	//
	Peeker		   : CollectionPeeker_Mock<5>;
	CollectionName : T_MaxString;
	i			   : UDINT;
END_VAR
IF TestSuite.Test(__POUNAME()).ExecuteTest() THEN
	Expected			  := TRUE;
	CollectionName		  := 'Test Collection';
	ExpectedNames[1]	  := ComponentArray[9].Name;
	ExpectedNames[2]	  := ComponentArray[0].Name;
	ExpectedNames[3]	  := ComponentArray[1].Name;
	ExpectedNames[4]	  := ComponentArray[2].Name;
	ExpectedNames[5]	  := ComponentArray[3].Name;
	Peeker.CollectionName := CollectionName;
	Peeker.PeekCollection(AllComponents);
	Peeker.MoveUpOne := TRUE;
	NamesEqual		 := TRUE;
	FOR i := 1 TO 5 DO
		__QUERYINTERFACE(Peeker.Items[i], CurrentComponent);
		ActualNames[i] := CurrentComponent.Name;
		NamesEqual	   := NamesEqual AND ActualNames[i] = ExpectedNames[i];
	END_FOR

	Actual := Peeker.FirstItem = 10 AND Peeker.LastItem = 4 AND NamesEqual;
	TestSuite.Test(__POUNAME()).AssertEqual(Expected, Actual);
END_IF
END_METHOD

METHOD NoCollection
VAR
	Expected : BOOL;
	Actual	 : BOOL;

	//
	Peeker		   : CollectionPeeker_Mock<5>;
	CollectionName : T_MaxString;
END_VAR
IF TestSuite.Test(__POUNAME()).ExecuteTest() THEN
	Expected		   := TRUE;
	CollectionName	   := '';
	Peeker.MoveDownOne := TRUE;
	Peeker.MoveUpOne   := TRUE;
	Peeker.PageDown	   := TRUE;
	Peeker.PageUp	   := TRUE;
	Actual			   := Peeker.CollectionName = CollectionName;
	TestSuite.Test(__POUNAME()).AssertEqual(Expected, Actual);
END_IF
END_METHOD

METHOD PageDownOne
VAR
	Expected		 : BOOL;
	Actual			 : BOOL;
	NamesEqual		 : BOOL;
	ExpectedNames	 : ARRAY[1..5] OF STRING[5];
	ActualNames		 : ARRAY[1..5] OF STRING[5];
	CurrentComponent : I_Component;

	//
	Peeker		   : CollectionPeeker_Mock<5>;
	CollectionName : T_MaxString;
	i			   : UDINT;
END_VAR
IF TestSuite.Test(__POUNAME()).ExecuteTest() THEN
	Expected			  := TRUE;
	CollectionName		  := 'Test Collection';
	ExpectedNames[1]	  := ComponentArray[5].Name;
	ExpectedNames[2]	  := ComponentArray[6].Name;
	ExpectedNames[3]	  := ComponentArray[7].Name;
	ExpectedNames[4]	  := ComponentArray[8].Name;
	ExpectedNames[5]	  := ComponentArray[9].Name;
	Peeker.CollectionName := CollectionName;
	Peeker.PeekCollection(AllComponents);
	Peeker.PageDown := TRUE;
	NamesEqual		:= TRUE;
	FOR i := 1 TO 5 DO
		__QUERYINTERFACE(Peeker.Items[i], CurrentComponent);
		ActualNames[i] := CurrentComponent.Name;
		NamesEqual	   := NamesEqual AND ActualNames[i] = ExpectedNames[i];
	END_FOR

	Actual := Peeker.FirstItem = 6 AND Peeker.LastItem = 10 AND NamesEqual;
	TestSuite.Test(__POUNAME()).AssertEqual(Expected, Actual);
END_IF
END_METHOD

METHOD PageDownRollover
VAR
	Expected		 : BOOL;
	Actual			 : BOOL;
	NamesEqual		 : BOOL;
	ExpectedNames	 : ARRAY[1..5] OF STRING[5];
	ActualNames		 : ARRAY[1..5] OF STRING[5];
	CurrentComponent : I_Component;

	//
	Peeker		   : CollectionPeeker_Mock<5>;
	CollectionName : T_MaxString;
	i			   : UDINT;
END_VAR
IF TestSuite.Test(__POUNAME()).ExecuteTest() THEN
	Expected			  := TRUE;
	CollectionName		  := 'Test Collection';
	ExpectedNames[1]	  := ComponentArray[8].Name;
	ExpectedNames[2]	  := ComponentArray[9].Name;
	ExpectedNames[3]	  := ComponentArray[0].Name;
	ExpectedNames[4]	  := ComponentArray[1].Name;
	ExpectedNames[5]	  := ComponentArray[2].Name;
	Peeker.CollectionName := CollectionName;
	Peeker.PeekCollection(AllComponents);
	Peeker.FirstItem := 4;
	Peeker.PageDown	 := TRUE;
	NamesEqual		 := TRUE;
	FOR i := 1 TO 5 DO
		__QUERYINTERFACE(Peeker.Items[i], CurrentComponent);
		ActualNames[i] := CurrentComponent.Name;
		NamesEqual	   := NamesEqual AND ActualNames[i] = ExpectedNames[i];
	END_FOR

	Actual := Peeker.FirstItem = 9 AND Peeker.LastItem = 3 AND NamesEqual;
	TestSuite.Test(__POUNAME()).AssertEqual(Expected, Actual);
END_IF
END_METHOD

METHOD PageUpOne
VAR
	Expected		 : BOOL;
	Actual			 : BOOL;
	NamesEqual		 : BOOL;
	ExpectedNames	 : ARRAY[1..5] OF STRING[5];
	ActualNames		 : ARRAY[1..5] OF STRING[5];
	CurrentComponent : I_Component;

	//
	Peeker		   : CollectionPeeker_Mock<5>;
	CollectionName : T_MaxString;
	i			   : UDINT;
END_VAR
IF TestSuite.Test(__POUNAME()).ExecuteTest() THEN
	Expected			  := TRUE;
	CollectionName		  := 'Test Collection';
	ExpectedNames[1]	  := ComponentArray[1].Name;
	ExpectedNames[2]	  := ComponentArray[2].Name;
	ExpectedNames[3]	  := ComponentArray[3].Name;
	ExpectedNames[4]	  := ComponentArray[4].Name;
	ExpectedNames[5]	  := ComponentArray[5].Name;
	Peeker.CollectionName := CollectionName;
	Peeker.PeekCollection(AllComponents);
	Peeker.FirstItem := 7;
	Peeker.PageUp	 := TRUE;
	NamesEqual		 := TRUE;
	FOR i := 1 TO 5 DO
		__QUERYINTERFACE(Peeker.Items[i], CurrentComponent);
		ActualNames[i] := CurrentComponent.Name;
		NamesEqual	   := NamesEqual AND ActualNames[i] = ExpectedNames[i];
	END_FOR

	Actual := Peeker.FirstItem = 2 AND Peeker.LastItem = 6 AND NamesEqual;
	TestSuite.Test(__POUNAME()).AssertEqual(Expected, Actual);
END_IF
END_METHOD

METHOD PageUpRollOver
VAR
	Expected		 : BOOL;
	Actual			 : BOOL;
	NamesEqual		 : BOOL;
	ExpectedNames	 : ARRAY[1..5] OF STRING[5];
	ActualNames		 : ARRAY[1..5] OF STRING[5];
	CurrentComponent : I_Component;

	//
	Peeker		   : CollectionPeeker_Mock<5>;
	CollectionName : T_MaxString;
	i			   : UDINT;
END_VAR
IF TestSuite.Test(__POUNAME()).ExecuteTest() THEN
	Expected			  := TRUE;
	CollectionName		  := 'Test Collection';
	ExpectedNames[1]	  := ComponentArray[6].Name;
	ExpectedNames[2]	  := ComponentArray[7].Name;
	ExpectedNames[3]	  := ComponentArray[8].Name;
	ExpectedNames[4]	  := ComponentArray[9].Name;
	ExpectedNames[5]	  := ComponentArray[0].Name;
	Peeker.CollectionName := CollectionName;
	Peeker.PeekCollection(AllComponents);
	Peeker.FirstItem := 2;
	Peeker.PageUp	 := TRUE;
	NamesEqual		 := TRUE;
	FOR i := 1 TO 5 DO
		__QUERYINTERFACE(Peeker.Items[i], CurrentComponent);
		ActualNames[i] := CurrentComponent.Name;
		NamesEqual	   := NamesEqual AND ActualNames[i] = ExpectedNames[i];
	END_FOR

	Actual := Peeker.FirstItem = 7 AND Peeker.LastItem = 1 AND NamesEqual;
	TestSuite.Test(__POUNAME()).AssertEqual(Expected, Actual);
END_IF
END_METHOD

METHOD SetCollectionCheck
VAR
	Expected		 : BOOL;
	Actual			 : BOOL;
	NamesEqual		 : BOOL;
	ExpectedNames	 : ARRAY[1..5] OF STRING[5];
	ActualNames		 : ARRAY[1..5] OF STRING[5];
	CurrentComponent : I_Component;

	//
	Peeker		   : CollectionPeeker_Mock<5>;
	CollectionName : T_MaxString;
	i			   : UDINT;
END_VAR
IF TestSuite.Test(__POUNAME()).ExecuteTest() THEN
	Expected			  := TRUE;
	CollectionName		  := 'Test Collection';
	ExpectedNames[1]	  := ComponentArray[0].Name;
	ExpectedNames[2]	  := ComponentArray[1].Name;
	ExpectedNames[3]	  := ComponentArray[2].Name;
	ExpectedNames[4]	  := ComponentArray[3].Name;
	ExpectedNames[5]	  := ComponentArray[4].Name;
	Peeker.CollectionName := CollectionName;
	Peeker.PeekCollection(AllComponents);
	NamesEqual := TRUE;
	FOR i := 1 TO 5 DO
		__QUERYINTERFACE(Peeker.Items[i], CurrentComponent);
		ActualNames[i] := CurrentComponent.Name;
		NamesEqual	   := NamesEqual AND ActualNames[i] = ExpectedNames[i];
	END_FOR

	Actual := Peeker.CollectionName = CollectionName AND Peeker.Collection.Count = AllComponents.Count AND Peeker.FirstItem = 1 AND Peeker.LastItem = 5 AND NamesEqual;
	TestSuite.Test(__POUNAME()).AssertEqual(Expected, Actual);
END_IF
END_METHOD

METHOD SetFirstItem
VAR
	Expected		 : BOOL;
	Actual			 : BOOL;
	NamesEqual		 : BOOL;
	ExpectedNames	 : ARRAY[1..5] OF STRING[5];
	ActualNames		 : ARRAY[1..5] OF STRING[5];
	CurrentComponent : I_Component;

	//
	Peeker		   : CollectionPeeker_Mock<5>;
	CollectionName : T_MaxString;
	i			   : UDINT;
END_VAR
IF TestSuite.Test(__POUNAME()).ExecuteTest() THEN
	Expected			  := TRUE;
	CollectionName		  := 'Test Collection';
	ExpectedNames[1]	  := ComponentArray[4].Name;
	ExpectedNames[2]	  := ComponentArray[5].Name;
	ExpectedNames[3]	  := ComponentArray[6].Name;
	ExpectedNames[4]	  := ComponentArray[7].Name;
	ExpectedNames[5]	  := ComponentArray[8].Name;
	Peeker.CollectionName := CollectionName;
	Peeker.PeekCollection(AllComponents);
	Peeker.FirstItem := 5;
	NamesEqual		 := TRUE;
	FOR i := 1 TO 5 DO
		__QUERYINTERFACE(Peeker.Items[i], CurrentComponent);
		ActualNames[i] := CurrentComponent.Name;
		NamesEqual	   := NamesEqual AND ActualNames[i] = ExpectedNames[i];
	END_FOR

	Actual := Peeker.FirstItem = 5 AND Peeker.LastItem = 9 AND NamesEqual;
	TestSuite.Test(__POUNAME()).AssertEqual(Expected, Actual);
END_IF
END_METHOD

END_FUNCTION_BLOCK

// ---- _Mockups/CollectionPeeker/CollectionPeeker_Mock.TcPOU
FUNCTION_BLOCK CollectionPeeker_Mock
VAR_GENERIC CONSTANT
	PeekSize2 : UDINT := 5;
END_VAR
EXTENDS CollectionPeeker<PeekSize2>
VAR
END_VAR

PROPERTY Collection : I_Collection
GET
Collection := _Collection;
END_GET
END_PROPERTY

END_FUNCTION_BLOCK

// ---- UnitTests/Force/ForcibleBool_TEST.TcPOU
FUNCTION_BLOCK ForcibleBool_TEST
VAR
END_VAR

ForceOff();
ForceOn();
UnforcedOff();
UnforcedOn();

METHOD ForceOff
VAR
	Expected	 : BOOL;
	Actual		 : BOOL;
	ForcibleBool : ForcibleBool('');
END_VAR
IF TestSuite.Test(__POUNAME()).ExecuteTest() THEN
	Expected := FALSE;
	ForcibleBool.SetForceState(E_ForceState.ForceOff);
	ForcibleBool.Input := TRUE;
	Actual			   := ForcibleBool.Output;
	TestSuite.Test(__POUNAME()).AssertEqual(Expected, Actual);
END_IF
END_METHOD

METHOD ForceOn
VAR
	Expected	 : BOOL;
	Actual		 : BOOL;
	ForcibleBool : ForcibleBool('');
END_VAR
IF TestSuite.Test(__POUNAME()).ExecuteTest() THEN
	Expected := TRUE;
	ForcibleBool.SetForceState(E_ForceState.ForceOn);
	ForcibleBool.Input := FALSE;
	Actual			   := ForcibleBool.Output;
	TestSuite.Test(__POUNAME()).AssertEqual(Expected, Actual);
END_IF
END_METHOD

METHOD UnforcedOff
VAR
	Expected	 : BOOL;
	Actual		 : BOOL;
	ForcibleBool : ForcibleBool('');
END_VAR
IF TestSuite.Test(__POUNAME()).ExecuteTest() THEN
	Expected := FALSE;
	ForcibleBool.SetForceState(E_ForceState.Unforced);
	ForcibleBool.Input := FALSE;
	Actual			   := ForcibleBool.Output;
	TestSuite.Test(__POUNAME()).AssertEqual(Expected, Actual);
END_IF
END_METHOD

METHOD UnforcedOn
VAR
	Expected	 : BOOL;
	Actual		 : BOOL;
	ForcibleBool : ForcibleBool('');
END_VAR
IF TestSuite.Test(__POUNAME()).ExecuteTest() THEN
	Expected := TRUE;
	ForcibleBool.SetForceState(E_ForceState.Unforced);
	ForcibleBool.Input := TRUE;
	Actual			   := ForcibleBool.Output;
	TestSuite.Test(__POUNAME()).AssertEqual(Expected, Actual);
END_IF
END_METHOD

END_FUNCTION_BLOCK

// ---- UnitTests/Force/ForcibleInt_Test.TcPOU
FUNCTION_BLOCK ForcibleInt_Test
VAR
END_VAR

ForceOff();
ForceOn();
ForcibleAcceptsValue();
ForciblePassesUnforcedValue();

METHOD ForceOff
VAR
	Expected	 : INT;
	Actual		 : INT;
	Forcible : ForcibleInt('');
END_VAR
IF TestSuite.Test(__POUNAME()).ExecuteTest() THEN
	Expected := 0;
	Forcible.SetForceState(E_ForceState.ForceOff);
	Forcible.Input := 12;
	Actual	:= Forcible.Output;
	TestSuite.Test(__POUNAME()).AssertEqual(Expected, Actual);
END_IF
END_METHOD

METHOD ForceOn
VAR
	Expected	 : INT;
	Actual		 : INT;
	Forcible : ForcibleInt('');
END_VAR
IF TestSuite.Test(__POUNAME()).ExecuteTest() THEN
	Expected := 16;
	Forcible.ForceValue := 16;
	Forcible.SetForceState(E_ForceState.ForceOn);
	Forcible.Input := 23;
	Actual			   := Forcible.Output;
	TestSuite.Test(__POUNAME()).AssertEqual(Expected, Actual);
END_IF
END_METHOD

METHOD ForcibleAcceptsValue
VAR
	Expected	 : INT;
	Actual		 : INT;
	Forcible : ForcibleInt('');
END_VAR
IF TestSuite.Test(__POUNAME()).ExecuteTest() THEN
	Expected := 17;
	Forcible.ForceValue := Expected;
	Actual			   := Forcible.ForceValue;
	TestSuite.Test(__POUNAME()).AssertEqual(Expected, Actual);
END_IF
END_METHOD

METHOD ForciblePassesUnforcedValue
VAR
	Expected	 : INT;
	Actual		 : INT;
	Forcible : ForcibleInt('');
END_VAR
IF TestSuite.Test(__POUNAME()).ExecuteTest() THEN
	Expected := 16;
	Forcible.SetForceState(E_ForceState.Unforced);
	Forcible.Input := 16;
	Actual			   := Forcible.Output;
	TestSuite.Test(__POUNAME()).AssertEqual(Expected, Actual);
END_IF
END_METHOD

END_FUNCTION_BLOCK

// ---- UnitTests/Utilities/Utilities_TEST.TcPOU
FUNCTION_BLOCK Utilities_TEST
VAR
END_VAR

CompareLREALFalse();
CompareLREALTrue();
CompareModuloFalse();
CompareModuloTrue();
PercentToAnalogConversion();
AnalogScaleReturns0IfInMinGTInMax();
AnalogScaleReturns0IfOutMinGTOutMax();
AnalogScaleReturnsOutMaxIFValueGTInMax();
AnalogScaleReturnsOutMinIFValueLTInMin();
AnalogueScaleConvertsCorrectly();
CalibrateAppliesGainCorrectly();
CalibrateAppliesOffsetCorrectly();

METHOD AnalogScaleReturns0IfInMinGTInMax
VAR
	InputGeneric : LREAL;
	TestScale : AnalogScale;

	Expected : LREAL := 0.0;
	Actual	 : LREAL;
END_VAR
IF TestSuite.Test(__POUNAME()).ExecuteTest() THEN
	InputGeneric							   := 750;
	TestScale.InputMaximum	   := 100;
	TestScale.InputMinimum	   := 200;
	TestScale.OutputMaximum	   := 10;
	TestScale.OutputMinimum	   := -10;
	Actual									   := TestScale.Transform(InputGeneric);
	TestSuite.Test(__POUNAME()).AssertEqual(Expected, Actual);
END_IF
END_METHOD

METHOD AnalogScaleReturns0IfOutMinGTOutMax
VAR
	InputGeneric : LREAL;
	TestScale : AnalogScale;

	Expected : LREAL := 0.0;
	Actual	 : LREAL;
END_VAR
IF TestSuite.Test(__POUNAME()).ExecuteTest() THEN
	InputGeneric							   := 750;
	TestScale.InputMaximum	   := 100;
	TestScale.InputMinimum	   := -200;
	TestScale.OutputMaximum	   := 10;
	TestScale.OutputMinimum	   := 20;
	Actual									   := TestScale.Transform(InputGeneric);
	TestSuite.Test(__POUNAME()).AssertEqual(Expected, Actual);
END_IF
END_METHOD

METHOD AnalogScaleReturnsOutMaxIFValueGTInMax
VAR
	InputGeneric : LREAL;
	TestScale : AnalogScale;

	Expected : LREAL := -10.0;
	Actual	 : LREAL;
END_VAR
IF TestSuite.Test(__POUNAME()).ExecuteTest() THEN
	InputGeneric			   := -110;
	TestScale.InputMaximum	   := 100;
	TestScale.InputMinimum	   := -100;
	TestScale.OutputMaximum	   := 10;
	TestScale.OutputMinimum	   := -10;
	Actual									   := TestScale.Transform(InputGeneric);
	TestSuite.Test(__POUNAME()).AssertEqual(Expected, Actual);
END_IF
END_METHOD

METHOD AnalogScaleReturnsOutMinIFValueLTInMin
VAR
	InputGeneric : LREAL;
	TestScale : AnalogScale;

	Expected : LREAL := 10.0;
	Actual	 : LREAL;
END_VAR
IF TestSuite.Test(__POUNAME()).ExecuteTest() THEN
	InputGeneric			   := 110;
	TestScale.InputMaximum	   := 100;
	TestScale.InputMinimum	   := -100;
	TestScale.OutputMaximum	   := 10;
	TestScale.OutputMinimum	   := -10;
	Actual									   := TestScale.Transform(InputGeneric);
	TestSuite.Test(__POUNAME()).AssertEqual(Expected, Actual);
END_IF
END_METHOD

METHOD AnalogueScaleConvertsCorrectly
VAR
	InputGeneric : LREAL;
	TestScale : AnalogScale;

	Expected : LREAL;
	Actual	 : LREAL;
END_VAR
IF TestSuite.Test(__POUNAME()).ExecuteTest() THEN
	InputGeneric							   := 500;
	Expected								   := 5;
	TestScale.InputMaximum	   := 1000;
	TestScale.InputMinimum	   := 0.0;
	TestScale.OutputMaximum	   := 10;
	TestScale.OutputMinimum	   := 0.0;
	Actual									   := TestScale.Transform(InputGeneric);
	TestSuite.Test(__POUNAME()).AssertEqual(Expected, Actual);
END_IF
END_METHOD

METHOD CalibrateAppliesGainCorrectly
VAR
	InputGeneric : LREAL;
	TestCalib : Calibrate;

	Expected : LREAL;
	Actual	 : LREAL;
END_VAR
IF TestSuite.Test(__POUNAME()).ExecuteTest() THEN
	InputGeneric							   := 500;
	Expected								   := 501;
	TestCalib.Gain	   := 1;
	TestCalib.Offset	   := 1.0;
	Actual									   := TestCalib.Transform(InputGeneric);
	TestSuite.Test(__POUNAME()).AssertEqual(Expected, Actual);
END_IF
END_METHOD

METHOD CalibrateAppliesOffsetCorrectly
VAR
	InputGeneric : LREAL;
	TestCalib : Calibrate;

	Expected : LREAL;
	Actual	 : LREAL;
END_VAR
IF TestSuite.Test(__POUNAME()).ExecuteTest() THEN
	InputGeneric							   := 500;
	Expected								   := 1000;
	TestCalib.Gain	   := 2;
	TestCalib.Offset	   := 0.0;
	Actual									   := TestCalib.Transform(InputGeneric);
	TestSuite.Test(__POUNAME()).AssertEqual(Expected, Actual);
END_IF
END_METHOD

METHOD CompareLREALFalse
VAR
	Expected : BOOL;
	Actual	 : BOOL;
END_VAR
IF TestSuite.Test(__POUNAME()).ExecuteTest() THEN
	Expected := FALSE;
	Actual	 := CompareLREAL(10.0, 11.8);
	TestSuite.Test(__POUNAME()).AssertEqual(Expected, Actual);
END_IF
END_METHOD

METHOD CompareLREALTrue
VAR
	Expected : BOOL;
	Actual	 : BOOL;
END_VAR
IF TestSuite.Test(__POUNAME()).ExecuteTest() THEN
	Expected := TRUE;
	Actual	 := CompareLREAL(10.5, 10.5);
	TestSuite.Test(__POUNAME()).AssertEqual(Expected, Actual);
END_IF
END_METHOD

METHOD CompareModuloFalse
VAR
	Expected : BOOL;
	Actual	 : BOOL;
END_VAR
IF TestSuite.Test(__POUNAME()).ExecuteTest() THEN
	Expected := FALSE;
	Actual	 := CompareModulo(360, 500);
	TestSuite.Test(__POUNAME()).AssertEqual(Expected, Actual);
END_IF
END_METHOD

METHOD CompareModuloTrue
VAR
	Expected : BOOL;
	Actual	 : BOOL;
END_VAR
IF TestSuite.Test(__POUNAME()).ExecuteTest() THEN
	Expected := TRUE;
	Actual	 := CompareModulo(0, 720);
	TestSuite.Test(__POUNAME()).AssertEqual(Expected, Actual);
END_IF
END_METHOD

METHOD PercentToAnalogConversion
VAR
	Expected : INT;
	Actual	 : INT;
END_VAR
IF TestSuite.Test(__POUNAME()).ExecuteTest() THEN
	Expected := 16383;
	Actual	 := PercentToAnalog(50);
	TestSuite.Test(__POUNAME()).AssertEqual(Expected, Actual);
END_IF
END_METHOD

END_FUNCTION_BLOCK

// ---- UnitTests/Digital/DigitalInput_NC_TEST.TcPOU
FUNCTION_BLOCK DigitalInput_NC_TEST
VAR
END_VAR

ForcedOn();
ForcedOff();
On();
Off();

METHOD ForcedOff : BOOL
VAR
	Expected		: BOOL;
	Actual			: BOOL;
	Input			: BOOL;
	DigitalInput_NC : DigitalInput_NC('DigitalInput', Input);
END_VAR
IF TestSuite.Test(__POUNAME()).ExecuteTest() THEN
	Expected			  := FALSE;
	DigitalInput_NC.Force := E_ForceState.ForceOff;
	Input				  := FALSE;
	Actual				  := DigitalInput_NC.IsActive;
	TestSuite.Test(__POUNAME()).AssertEqual(Expected, Actual);
END_IF
END_METHOD

METHOD ForcedOn : BOOL
VAR
	Expected		: BOOL;
	Actual			: BOOL;
	Input			: BOOL;
	DigitalInput_NC : DigitalInput_NC('DigitalInput', Input);
END_VAR
IF TestSuite.Test(__POUNAME()).ExecuteTest() THEN
	Expected			  := TRUE;
	DigitalInput_NC.Force := E_ForceState.ForceOn;
	Input				  := TRUE;
	Actual				  := DigitalInput_NC.IsActive;
	TestSuite.Test(__POUNAME()).AssertEqual(Expected, Actual);
END_IF
END_METHOD

METHOD Off : BOOL
VAR
	Expected		: BOOL;
	Actual			: BOOL;
	Input			: BOOL;
	DigitalInput_NC : DigitalInput_NC('DigitalInput', Input);
END_VAR
IF TestSuite.Test(__POUNAME()).ExecuteTest() THEN
	Expected			  := FALSE;
	DigitalInput_NC.Force := E_ForceState.Unforced;
	Input				  := TRUE;
	Actual				  := DigitalInput_NC.IsActive;
	TestSuite.Test(__POUNAME()).AssertEqual(Expected, Actual);
END_IF
END_METHOD

METHOD On
VAR
	Expected		: BOOL;
	Actual			: BOOL;
	Input			: BOOL;
	DigitalInput_NC : DigitalInput_NC('DigitalInput', Input);
END_VAR
IF TestSuite.Test(__POUNAME()).ExecuteTest() THEN
	Expected			  := TRUE;
	DigitalInput_NC.Force := E_ForceState.Unforced;
	Input				  := FALSE;
	Actual				  := DigitalInput_NC.IsActive;
	TestSuite.Test(__POUNAME()).AssertEqual(Expected, Actual);
END_IF
END_METHOD

END_FUNCTION_BLOCK

// ---- UnitTests/Digital/DigitalInput_NO_TEST.TcPOU
FUNCTION_BLOCK DigitalInput_NO_TEST
VAR
END_VAR

ForcedOn();
ForcedOff();
On();
Off();

METHOD ForcedOff : BOOL
VAR
	Expected		: BOOL;
	Actual			: BOOL;
	Input			: BOOL;
	DigitalInput_NO : DigitalInput_NO('DigitalInput', Input);
END_VAR
IF TestSuite.Test(__POUNAME()).ExecuteTest() THEN
	Expected			  := FALSE;
	DigitalInput_NO.Force := E_ForceState.ForceOff;
	Input				  := TRUE;
	Actual				  := DigitalInput_NO.IsActive;
	TestSuite.Test(__POUNAME()).AssertEqual(Expected, Actual);
END_IF
END_METHOD

METHOD ForcedOn : BOOL
VAR
	Expected		: BOOL;
	Actual			: BOOL;
	Input			: BOOL;
	DigitalInput_NO : DigitalInput_NO('DigitalInput', Input);
END_VAR
IF TestSuite.Test(__POUNAME()).ExecuteTest() THEN
	Expected			  := TRUE;
	DigitalInput_NO.Force := E_ForceState.ForceOn;
	Input				  := FALSE;
	Actual				  := DigitalInput_NO.IsActive;
	TestSuite.Test(__POUNAME()).AssertEqual(Expected, Actual);
END_IF
END_METHOD

METHOD Off : BOOL
VAR
	Expected		: BOOL;
	Actual			: BOOL;
	Input			: BOOL;
	DigitalInput_NO : DigitalInput_NO('DigitalInput', Input);
END_VAR
IF TestSuite.Test(__POUNAME()).ExecuteTest() THEN
	Expected			  := FALSE;
	DigitalInput_NO.Force := E_ForceState.Unforced;
	Input				  := FALSE;
	Actual				  := DigitalInput_NO.IsActive;
	TestSuite.Test(__POUNAME()).AssertEqual(Expected, Actual);
END_IF
END_METHOD

METHOD On
VAR
	Expected		: BOOL;
	Actual			: BOOL;
	Input			: BOOL;
	DigitalInput_NO : DigitalInput_NO('DigitalInput', Input);
END_VAR
IF TestSuite.Test(__POUNAME()).ExecuteTest() THEN
	Expected			  := TRUE;
	DigitalInput_NO.Force := E_ForceState.Unforced;
	Input				  := TRUE;
	Actual				  := DigitalInput_NO.IsActive;
	TestSuite.Test(__POUNAME()).AssertEqual(Expected, Actual);
END_IF
END_METHOD

END_FUNCTION_BLOCK

// ---- UnitTests/Digital/DigitalOutput_TEST.TcPOU
FUNCTION_BLOCK DigitalOutput_TEST
VAR
END_VAR

ForcedOn();
ForcedOff();
On();
Off();
ForceOffVisitor();
ForceOnVisitor();

METHOD ForcedOff
VAR
	Expected	  : BOOL;
	Actual		  : BOOL;
	Output		  : BOOL;
	DigitalOutput : DigitalOutput('Name', Output);
END_VAR
IF TestSuite.Test(__POUNAME()).ExecuteTest() THEN
	Expected			:= FALSE;
	DigitalOutput.Force := E_ForceState.ForceOff;
	DigitalOutput.On	:= TRUE;
	Actual				:= Output;
	TestSuite.Test(__POUNAME()).AssertEqual(Expected, Actual);
END_IF
END_METHOD

METHOD ForcedOn
VAR
	Expected	  : BOOL;
	Actual		  : BOOL;
	Output		  : BOOL;
	DigitalOutput : DigitalOutput('Name', Output);
END_VAR
IF TestSuite.Test(__POUNAME()).ExecuteTest() THEN
	Expected			:= TRUE;
	DigitalOutput.Force := E_ForceState.ForceOn;
	DigitalOutput.On	:= FALSE;
	Actual				:= Output;
	TestSuite.Test(__POUNAME()).AssertEqual(Expected, Actual);
END_IF
END_METHOD

METHOD ForceOffVisitor
VAR
	Expected	  : BOOL;
	Actual		  : BOOL;
	Output		  : BOOL;
	DigitalOutput : DigitalOutput('Name', Output);
	ForceVisitor  : ForceVisitor;
END_VAR
IF TestSuite.Test(__POUNAME()).ExecuteTest() THEN
	Expected			:= FALSE;
	DigitalOutput.Force := E_ForceState.ForceOn;
	ForceVisitor.Force	:= E_ForceState.ForceOff;
	DigitalOutput.Accept(ForceVisitor);
	DigitalOutput.On := TRUE;
	Actual			 := Output;
	TestSuite.Test(__POUNAME()).AssertEqual(Expected, Actual);
END_IF
END_METHOD

METHOD ForceOnVisitor
VAR
	Expected	  : BOOL;
	Actual		  : BOOL;
	Output		  : BOOL;
	DigitalOutput : DigitalOutput('Name', Output);
	ForceVisitor  : ForceVisitor;
END_VAR
IF TestSuite.Test(__POUNAME()).ExecuteTest() THEN
	Expected			:= TRUE;
	DigitalOutput.Force := E_ForceState.ForceOff;
	ForceVisitor.Force	:= E_ForceState.ForceOn;
	DigitalOutput.Accept(ForceVisitor);
	DigitalOutput.On := FALSE;
	Actual			 := Output;
	TestSuite.Test(__POUNAME()).AssertEqual(Expected, Actual);
END_IF
END_METHOD

METHOD Off : BOOL
VAR
	Expected	  : BOOL;
	Actual		  : BOOL;
	Output		  : BOOL;
	DigitalOutput : DigitalOutput('Name', Output);
END_VAR
IF TestSuite.Test(__POUNAME()).ExecuteTest() THEN
	Expected			:= FALSE;
	DigitalOutput.Force := E_ForceState.Unforced;
	DigitalOutput.On	:= FALSE;
	Actual				:= Output;
	TestSuite.Test(__POUNAME()).AssertEqual(Expected, Actual);
END_IF
END_METHOD

METHOD On
VAR
	Expected	  : BOOL;
	Actual		  : BOOL;
	Output		  : BOOL;
	DigitalOutput : DigitalOutput('Name', Output);
END_VAR
IF TestSuite.Test(__POUNAME()).ExecuteTest() THEN
	Expected			:= TRUE;
	DigitalOutput.Force := E_ForceState.Unforced;
	DigitalOutput.On	:= TRUE;
	Actual				:= Output;
	TestSuite.Test(__POUNAME()).AssertEqual(Expected, Actual);
END_IF
END_METHOD

END_FUNCTION_BLOCK

// ---- UnitTests/Digital/DigitalInput_Combiner_TEST.TcPOU
FUNCTION_BLOCK DigitalInput_Combiner_TEST
VAR
END_VAR

AddTwoInputsBothActiveCheckIsActive();
AddTwoInputsOneActiveCheckIsActiveFalse();
CheckIsActiveFalseWhenNoInputAdded();
TryAddDuplicateInput();

METHOD AddTwoInputsBothActiveCheckIsActive
VAR
	Expected			  : BOOL;
	Actual				  : BOOL;
	Input1				  : BOOL;
	Input2				  : BOOL;
	DigitalInput1		  : DigitalInput_NO('Input1', Input1);
	DigitalInput2		  : DigitalInput_NO('Input2', Input2);
	DigitalInput_Combiner : DigitalInput_Combiner<2>('Input1 & Input2');
END_VAR
IF TestSuite.Test(__POUNAME()).ExecuteTest() THEN
	Expected := TRUE;
	Input1	 := TRUE;
	Input2	 := TRUE;
	DigitalInput_Combiner.AddInput(DigitalInput1);
	DigitalInput_Combiner.AddInput(DigitalInput2);
	Actual := DigitalInput_Combiner.IsActive;
	TestSuite.Test(__POUNAME()).AssertEqual(Expected, Actual);
END_IF
END_METHOD

METHOD AddTwoInputsOneActiveCheckIsActiveFalse
VAR
	Expected			  : BOOL;
	Actual				  : BOOL;
	Input1				  : BOOL;
	Input2				  : BOOL;
	DigitalInput1		  : DigitalInput_NO('Input1', Input1);
	DigitalInput2		  : DigitalInput_NO('Input2', Input2);
	DigitalInput_Combiner : DigitalInput_Combiner<2>('Input1 & Input2');
END_VAR
IF TestSuite.Test(__POUNAME()).ExecuteTest() THEN
	Expected := FALSE;
	Input1	 := FALSE;
	Input2	 := TRUE;
	DigitalInput_Combiner.AddInput(DigitalInput1);
	DigitalInput_Combiner.AddInput(DigitalInput2);
	Actual := DigitalInput_Combiner.IsActive;
	TestSuite.Test(__POUNAME()).AssertEqual(Expected, Actual);
END_IF
END_METHOD

METHOD CheckIsActiveFalseWhenNoInputAdded
VAR
	Expected			  : BOOL;
	Actual				  : BOOL;
	DigitalInput_Combiner : DigitalInput_Combiner<2>('Input1 & Input2');
END_VAR
IF TestSuite.Test(__POUNAME()).ExecuteTest() THEN
	Expected := FALSE;
	Actual	 := DigitalInput_Combiner.IsActive;
	TestSuite.Test(__POUNAME()).AssertEqual(Expected, Actual);
END_IF
END_METHOD

METHOD TryAddDuplicateInput
VAR
	Expected			  : BOOL;
	Actual				  : BOOL;
	Input1				  : BOOL;
	Input2				  : BOOL;
	DigitalInput1		  : DigitalInput_NO('Input1', Input1);
	DigitalInput2		  : DigitalInput_NO('Input2', Input2);
	DigitalInput_Combiner : DigitalInput_Combiner<2>('Input1 & Input2');
END_VAR
IF TestSuite.Test(__POUNAME()).ExecuteTest() THEN
	Expected := FALSE;
	Input1	 := TRUE;
	Input2	 := FALSE;
	DigitalInput_Combiner.AddInput(DigitalInput1);
	DigitalInput_Combiner.AddInput(DigitalInput1);
	DigitalInput_Combiner.AddInput(DigitalInput2);
	Actual := DigitalInput_Combiner.IsActive;
	TestSuite.Test(__POUNAME()).AssertEqual(Expected, Actual);
END_IF
END_METHOD

END_FUNCTION_BLOCK

// ---- UnitTests/Digital/DigitalInput_Debounce_TEST.TcPOU
FUNCTION_BLOCK DigitalInput_Debounce_TEST
// DebounceRisingEdgeOn
VAR
	RisingEdgeOnExpected						: BOOL;
	RisingEdgeOnActual							: BOOL;
	RisingEdgeOnInput1							: BOOL;
	RisingEdgeOnDigitalInput1					: DigitalInput_NO('Input1', RisingEdgeOnInput1);
	RisingEdgeOnDigitalInput_DebounceRisingEdge : DigitalInput_DebounceRisingEdge('Input1', RisingEdgeOnDigitalInput1);
	RisingEdgeOnTestTimer						: TON;
END_VAR

// DebounceRisingEdgeStayOff
VAR
	RisingEdgeStayOffExpected						 : BOOL;
	RisingEdgeStayOffActual							 : BOOL;
	RisingEdgeStayOffInput1							 : BOOL;
	RisingEdgeStayOffDigitalInput1					 : DigitalInput_NO('Input1', RisingEdgeStayOffInput1);
	RisingEdgeStayOffDigitalInput_DebounceRisingEdge : DigitalInput_DebounceRisingEdge('Input1', RisingEdgeStayOffDigitalInput1);
	RisingEdgeStayOffTestTimer						 : TON;
END_VAR

// DebounceFallingEdgeOn
VAR
	FallingEdgeOnExpected						  : BOOL;
	FallingEdgeOnActual							  : BOOL;
	FallingEdgeOnInput1							  : BOOL := TRUE;
	FallingEdgeOnDigitalInput1					  : DigitalInput_NO('Input1', FallingEdgeOnInput1);
	FallingEdgeOnDigitalInput_DebounceFallingEdge : DigitalInput_DebounceFallingEdge('Input1', FallingEdgeOnDigitalInput1);
	FallingEdgeOnTestTimer						  : TON;
END_VAR

// DebounceFallingEdgeStayOff
VAR
	FallingEdgeStayOffExpected						   : BOOL;
	FallingEdgeStayOffActual						   : BOOL;
	FallingEdgeStayOffInput1						   : BOOL := TRUE;
	FallingEdgeStayOffDigitalInput1					   : DigitalInput_NO('Input1', FallingEdgeStayOffInput1);
	FallingEdgeStayOffDigitalInput_DebounceFallingEdge : DigitalInput_DebounceFallingEdge('Input1', FallingEdgeStayOffDigitalInput1);
	FallingEdgeStayOffTestTimer						   : TON;
END_VAR

DebounceRisingEdgeStayOff();
DebounceRisingEdgeOn();
DebounceFallingEdgeStayOff();
DebounceFallingEdgeOn();

METHOD DebounceFallingEdgeOn
VAR_INPUT
END_VAR
IF TestSuite.Test(__POUNAME()).ExecuteTest() THEN
	FallingEdgeOnExpected := TRUE;

	//
	FallingEdgeOnDigitalInput_DebounceFallingEdge.DebounceTime := T#250MS;
	FallingEdgeOnDigitalInput_DebounceFallingEdge.CyclicLogic();
	FallingEdgeOnInput1 := FALSE;

	//
	FallingEdgeOnTestTimer(IN := TRUE, PT := T#235MS);
	IF FallingEdgeOnTestTimer.Q THEN
		FallingEdgeOnActual := FallingEdgeOnDigitalInput_DebounceFallingEdge.IsActive;
		TestSuite.Test(__POUNAME()).AssertEqual(FallingEdgeOnExpected, FallingEdgeOnActual);
	END_IF
END_IF
END_METHOD

METHOD DebounceFallingEdgeStayOff
VAR_INPUT
END_VAR
IF TestSuite.Test(__POUNAME()).ExecuteTest() THEN
	FallingEdgeStayOffExpected := FALSE;

	//
	FallingEdgeStayOffDigitalInput_DebounceFallingEdge.DebounceTime := T#250MS;
	FallingEdgeStayOffDigitalInput_DebounceFallingEdge.CyclicLogic();
	FallingEdgeStayOffInput1 := FALSE;

	//
	FallingEdgeStayOffTestTimer(IN := TRUE, PT := T#265MS);
	IF FallingEdgeStayOffTestTimer.Q THEN
		FallingEdgeStayOffActual := FallingEdgeStayOffDigitalInput_DebounceFallingEdge.IsActive;
		TestSuite.Test(__POUNAME()).AssertEqual(FallingEdgeStayOffExpected, FallingEdgeStayOffActual);
	END_IF
END_IF
END_METHOD

METHOD DebounceRisingEdgeOn
IF TestSuite.Test(__POUNAME()).ExecuteTest() THEN
	RisingEdgeOnExpected := TRUE;
	RisingEdgeOnInput1	 := TRUE;

	//
	RisingEdgeOnDigitalInput_DebounceRisingEdge.DebounceTime := T#250MS;
	RisingEdgeOnDigitalInput_DebounceRisingEdge.CyclicLogic();

	//
	RisingEdgeOnTestTimer(IN := TRUE, PT := T#250MS);
	IF RisingEdgeOnTestTimer.Q THEN
		RisingEdgeOnActual := RisingEdgeOnDigitalInput_DebounceRisingEdge.IsActive;
		TestSuite.Test(__POUNAME()).AssertEqual(RisingEdgeOnExpected, RisingEdgeOnActual);
	END_IF
END_IF
END_METHOD

METHOD DebounceRisingEdgeStayOff
VAR_INPUT
END_VAR
IF TestSuite.Test(__POUNAME()).ExecuteTest() THEN
	RisingEdgeStayOffExpected := FALSE;
	RisingEdgeStayOffInput1	  := TRUE;

	//
	RisingEdgeStayOffDigitalInput_DebounceRisingEdge.DebounceTime := T#250MS;
	RisingEdgeStayOffDigitalInput_DebounceRisingEdge.CyclicLogic();

	//
	RisingEdgeStayOffTestTimer(IN := TRUE, PT := T#235MS);
	IF RisingEdgeStayOffTestTimer.Q THEN
		RisingEdgeStayOffActual := RisingEdgeStayOffDigitalInput_DebounceRisingEdge.IsActive;
		TestSuite.Test(__POUNAME()).AssertEqual(RisingEdgeStayOffExpected, RisingEdgeStayOffActual);
	END_IF
END_IF
END_METHOD

END_FUNCTION_BLOCK

// ---- UnitTests/Cylinder/Cylinder_TEST.TcPOU
FUNCTION_BLOCK Cylinder_TEST
VAR
	DiExtended		   : BOOL;
	DiRetracted		   : BOOL;
	DoExtend		   : BOOL;
	DoRetract		   : BOOL;
	Extend			   : DigitalOutput('Extend', DoExtend);
	Retract			   : DigitalOutput('Retract', DoRetract);
	Extended		   : DigitalInput_NO('Extended', DiExtended);
	Retracted		   : DigitalInput_NO('Retracted', DiRetracted);
	TestCylinder	   : Cylinder('Test Cylinder', Extend, Retract, Extended, Retracted) := (ExtendTimeout := T#250MS, RetractTimeout := T#250MS);
	TestCylinderEvents : Cylinder_TcEvents('Test Cylinder Events', TestCylinder);
	TonTimeout		   : TON;
END_VAR

RetractCheckRetracting();
RetractCheckRetracted();
ExtendCheckExtending();
ExtendCheckExtended();
ErrorBothSensorsOn();
ErrorRetracting();
ErrorExtending();

METHOD ErrorBothSensorsOn
VAR
	Expected : DINT;
	Actual	 : DINT;
END_VAR
IF TestSuite.Test(__POUNAME()).ExecuteTest() THEN
	Expected	:= 3;
	DiRetracted := TRUE;
	DiExtended	:= TRUE;
	TestCylinder.CyclicLogic();
	TestCylinderEvents.CyclicLogic();
	Actual := TestCylinderEvents.GetHighestActiveEventReaction();
	TestSuite.Test(__POUNAME()).AssertEqual(Expected, Actual);

	// Cleanup
	DiRetracted := FALSE;
	DiExtended	:= FALSE;
	TestCylinder.Reset();
	TestCylinderEvents.Reset();
	TestCylinder.CyclicLogic();
	TestCylinderEvents.CyclicLogic();
END_IF
END_METHOD

METHOD ErrorExtending
VAR
	Expected : DINT;
	Actual	 : DINT;
END_VAR
IF TestSuite.Test(__POUNAME()).ExecuteTest() THEN
	Expected	:= 3;
	DiRetracted := FALSE;
	DiExtended	:= FALSE;
	TestCylinder.Extend();
	TestCylinderEvents.CyclicLogic();
	TestCylinder.CyclicLogic();
	TonTimeout.IN := TRUE;
	IF TonTimeout.Q THEN
		Actual := TestCylinderEvents.GetHighestActiveEventReaction();
		TestSuite.Test(__POUNAME()).AssertEqual(Expected, Actual);

		// Cleanup
		TonTimeout.IN := FALSE;
		DiExtended	  := TRUE;
		TestCylinder.Reset();
		TestCylinderEvents.Reset();
		TestCylinderEvents.CyclicLogic();
		TestCylinder.CyclicLogic();
	END_IF
END_IF

TonTimeout(PT := T#300MS);
END_METHOD

METHOD ErrorRetracting
VAR
	Expected : DINT;
	Actual	 : DINT;
END_VAR
IF TestSuite.Test(__POUNAME()).ExecuteTest() THEN
	Expected	:= 3;
	DiRetracted := FALSE;
	DiExtended	:= FALSE;
	TestCylinder.Retract();
	TestCylinder.CyclicLogic();
	TestCylinderEvents.CyclicLogic();
	TonTimeout.IN := TRUE;
	IF TonTimeout.Q THEN
		Actual := TestCylinderEvents.GetHighestActiveEventReaction();
		TestSuite.Test(__POUNAME()).AssertEqual(Expected, Actual);

		// Cleanup
		TonTimeout.IN := FALSE;
		DiRetracted	  := TRUE;
		TestCylinder.Reset();
		TestCylinderEvents.Reset();
		TestCylinderEvents.CyclicLogic();
		TestCylinder.CyclicLogic();
	END_IF
END_IF

TonTimeout(PT := T#300MS);
END_METHOD

METHOD ExtendCheckExtended
VAR
	Expected : BOOL;
	Actual	 : BOOL;
END_VAR
IF TestSuite.Test(__POUNAME()).ExecuteTest() THEN
	Expected	:= TRUE;
	DiRetracted := FALSE;
	DiExtended	:= TRUE;
	TestCylinder.CyclicLogic();
	Actual := TestCylinder.Extended;
	TestSuite.Test(__POUNAME()).AssertEqual(Expected, Actual);
END_IF
END_METHOD

METHOD ExtendCheckExtending
VAR
	Expected : BOOL;
	Actual	 : BOOL;
END_VAR
IF TestSuite.Test(__POUNAME()).ExecuteTest() THEN
	Expected := TRUE;
	TestCylinder.Extend();
	TestCylinder.CyclicLogic();
	Actual := TestCylinder.Extending;
	TestSuite.Test(__POUNAME()).AssertEqual(Expected, Actual);
END_IF
END_METHOD

METHOD RetractCheckRetracted
VAR
	Expected : BOOL;
	Actual	 : BOOL;
END_VAR
IF TestSuite.Test(__POUNAME()).ExecuteTest() THEN
	Expected	:= TRUE;
	DiRetracted := TRUE;
	TestCylinder.CyclicLogic();
	Actual := TestCylinder.Retracted;
	TestSuite.Test(__POUNAME()).AssertEqual(Expected, Actual);
END_IF
END_METHOD

METHOD RetractCheckRetracting
VAR
	Expected : BOOL;
	Actual	 : BOOL;
END_VAR
IF TestSuite.Test(__POUNAME()).ExecuteTest() THEN
	Expected := TRUE;
	TestCylinder.Retract();
	TestCylinder.CyclicLogic();
	Actual := TestCylinder.Retracting;
	TestSuite.Test(__POUNAME()).AssertEqual(Expected, Actual);
END_IF
END_METHOD

END_FUNCTION_BLOCK

// ---- UnitTests/Safety/SafetyBase_TEST.TcPOU
FUNCTION_BLOCK SafetyBase_TEST
VAR
	ResetPulse : SafetyResetPulse('Reset');
	Group	   : SafetyGroup_TcEvents('Group');
	EStop_Sim  : SafetyEstopFB_TcEvents('E-Stop');
	EStop_OK   : SafetyEstopFB_TcEvents('E-Stop') := (ResetFunction := ResetPulse);
	EStop_NOK  : SafetyEstopFB_TcEvents('E-Stop') := (ResetFunction := ResetPulse);
END_VAR

VAR
	Init				  : BOOL := TRUE;
	InfoData_Group AT %Q* : ST_SafetyStateDiag;
	InfoData_OK	   AT %Q* : ST_SafetyStateDiag;
	InfoData_NOK   AT %Q* : ST_SafetyStateDiag;
	Run			   AT %I* : BOOL;
	Reset		   AT %I* : BOOL;
END_VAR

IF Init THEN
	InfoData_Group.State := E_SafetyGroup_State.Run;
	InfoData_OK.State	 := E_SafetyEStop_State.Run;
	InfoData_NOK.State	 := E_SafetyEStop_State.Error;
	Init				 := FALSE;
ELSE
	Group.CyclicLogic();
	EStop_OK.CyclicLogic();
	EStop_NOK.CyclicLogic();
	SimEstopOK();
	SimEstopOK();
	EstopOK();
	EstopNOK();
	GroupRun();
	EstopReset();
END_IF

METHOD EstopNOK
VAR_INST
	Expected : BOOL;
	Actual	 : BOOL;
END_VAR
IF TestSuite.Test(__POUNAME()).ExecuteTest() THEN
	Expected := FALSE;
	Actual	 := EStop_NOK.OK;
	TestSuite.Test(__POUNAME()).AssertEqual(Expected, Actual);
END_IF
END_METHOD

METHOD EstopOK
VAR_INST
	Expected : BOOL;
	Actual	 : BOOL;
END_VAR
IF TestSuite.Test(__POUNAME()).ExecuteTest() THEN
	Expected := TRUE;
	Actual	 := EStop_OK.OK;
	TestSuite.Test(__POUNAME()).AssertEqual(Expected, Actual);
END_IF
END_METHOD

METHOD EstopReset
VAR_INST
	Expected  : BOOL;
	Actual	  : BOOL;
	TestDelay : TON;
END_VAR
IF TestSuite.Test(__POUNAME()).ExecuteTest() THEN
	TestDelay(IN := TRUE, PT := T#50MS);
	Expected := TRUE;
	EStop_NOK.Reset();
	IF TestDelay.Q THEN
		Actual := Reset;
		TestSuite.Test(__POUNAME()).AssertEqual(Expected, Actual);
	END_IF
END_IF
END_METHOD

METHOD GroupRun
VAR_INST
	Expected : BOOL;
	Actual	 : BOOL;
END_VAR
IF TestSuite.Test(__POUNAME()).ExecuteTest() THEN
	Expected := TRUE;
	Actual	 := Run;
	TestSuite.Test(__POUNAME()).AssertEqual(Expected, Actual);
END_IF
END_METHOD

METHOD SimEstopNOK
VAR_INST
	Expected : BOOL;
	Actual	 : BOOL;
END_VAR
IF TestSuite.Test(__POUNAME()).ExecuteTest() THEN
	Expected := FALSE;
	EStop_Sim.SimulateSafetyState(E_SafetyEStop_State.Error);
	EStop_Sim.CyclicLogic();
	Actual := EStop_Sim.OK;
	TestSuite.Test(__POUNAME()).AssertEqual(Expected, Actual);
END_IF
END_METHOD

METHOD SimEstopOK
VAR_INST
	Expected : BOOL;
	Actual	 : BOOL;
END_VAR
IF TestSuite.Test(__POUNAME()).ExecuteTest() THEN
	Expected := TRUE;
	EStop_Sim.SimulateSafetyState(E_SafetyEStop_State.Run);
	EStop_Sim.CyclicLogic();
	Actual := EStop_Sim.OK;
	TestSuite.Test(__POUNAME()).AssertEqual(Expected, Actual);
END_IF
END_METHOD

END_FUNCTION_BLOCK

// ---- UnitTests/ADS/ADS_TEST.TcPOU
FUNCTION_BLOCK ADS_TEST
VAR
	AdsReadWrite		: AdsReadWrite('Ads Read/Write') := (AmsNetId := '', AmsPort := 851);
	AdsRwNumber AT %MD0 : UDINT							 := 50;
	AdsRwSymbol			: UDINT							 := 85;
	Value				: UDINT;
END_VAR

AdsRead();
AdsWrite();
AdsReadBySymbol();
AdsWriteBySymbol();
AdsReadWrite.CyclicLogic();

METHOD AdsRead
VAR_INST
	Expected : UDINT;
	Actual	 : UDINT;
	Seq		 : UDINT;
END_VAR
IF TestSuite.Test(__POUNAME()).ExecuteTest() THEN
	Expected := AdsRwNumber;
	CASE Seq OF
		0:
			AdsReadWrite.Read(IdxGrp	:= 16#4020,
							  IdxOffset := 16#0,
							  pDestAddr := ADR(Value),
							  Length	:= SIZEOF(Value));

			Seq := 10;

		10:
			IF NOT AdsReadWrite.Busy THEN
				Seq := 20;
			END_IF

		20:
			Actual := Value;
			TestSuite.Test(__POUNAME()).AssertEqual(Expected, Actual);
	END_CASE
END_IF
END_METHOD

METHOD AdsReadBySymbol
VAR_INST
	Expected : UDINT;
	Actual	 : UDINT;
	Seq		 : UDINT;
END_VAR
IF TestSuite.Test(__POUNAME()).ExecuteTest() THEN
	Expected := AdsRwSymbol;
	CASE Seq OF
		0:
			AdsReadWrite.ReadBySymbol(SymbolName := 'TestsBase.ADS_TEST.AdsRwSymbol', pDestAddr := ADR(Value), Length := SIZEOF(Value));
			Seq := 10;

		10:
			IF NOT AdsReadWrite.Busy THEN
				Seq := 20;
			END_IF

		20:
			Actual := Value;
			TestSuite.Test(__POUNAME()).AssertEqual(Expected, Actual);
	END_CASE
END_IF
END_METHOD

METHOD AdsWrite
VAR_INST
	Expected : UDINT;
	Actual	 : UDINT;
	Seq		 : UDINT;
END_VAR
IF TestSuite.Test(__POUNAME()).ExecuteTest() THEN
	Expected := 95;
	CASE Seq OF
		0:
			Value := 95;
			AdsReadWrite.Write(IdxGrp	   := 16#4020,
							   IdxOffset   := 16#0,
							   pSourceAddr := ADR(Value),
							   Length	   := SIZEOF(Value));

			Seq := 10;

		10:
			IF NOT AdsReadWrite.Busy THEN
				Seq := 20;
			END_IF

		20:
			Actual := AdsRwNumber;
			TestSuite.Test(__POUNAME()).AssertEqual(Expected, Actual);
	END_CASE
END_IF
END_METHOD

METHOD AdsWriteBySymbol
VAR_INST
	Expected : UDINT;
	Actual	 : UDINT;
	Seq		 : UDINT;
END_VAR
IF TestSuite.Test(__POUNAME()).ExecuteTest() THEN
	Expected := 79;
	CASE Seq OF
		0:
			Value := 79;
			AdsReadWrite.WriteBySymbol(SymbolName := 'TestsBase.ADS_TEST.AdsRwSymbol', pSourceAddr := ADR(Value), Length := SIZEOF(Value));
			Seq := 10;

		10:
			IF NOT AdsReadWrite.Busy THEN
				Seq := 20;
			END_IF

		20:
			Actual := AdsRwSymbol;
			TestSuite.Test(__POUNAME()).AssertEqual(Expected, Actual);
	END_CASE
END_IF
END_METHOD

END_FUNCTION_BLOCK

// ---- UnitTests/Digital/DigitalInput_ForceVisitor_TEST.TcPOU
FUNCTION_BLOCK DigitalInput_ForceVisitor_TEST
VAR
END_VAR

ForceOffVisitor_NO();
ForceOnVisitor_NO();
UnforcedVisitor_NO();
ForceOffVisitor_NC();
ForceOnVisitor_NC();
UnforcedVisitor_NC();

METHOD ForceOffVisitor_NC
VAR
	Expected	 : BOOL;
	Actual		 : BOOL;
	Input		 : BOOL;
	DigitalInput : DigitalInput_NC('DigitalInput', Input);
	ForceVisitor : ForceVisitor;
END_VAR
IF TestSuite.Test(__POUNAME()).ExecuteTest() THEN
	Expected		   := FALSE;
	DigitalInput.Force := E_ForceState.ForceOn;
	ForceVisitor.Force := E_ForceState.ForceOff;
	DigitalInput.Accept(ForceVisitor);
	Input  := FALSE;
	Actual := DigitalInput.IsActive;
	TestSuite.Test(__POUNAME()).AssertEqual(Expected, Actual);
END_IF
END_METHOD

METHOD ForceOffVisitor_NO
VAR
	Expected	 : BOOL;
	Actual		 : BOOL;
	Input		 : BOOL;
	DigitalInput : DigitalInput_NO('DigitalInput', Input);
	ForceVisitor : ForceVisitor;
END_VAR
IF TestSuite.Test(__POUNAME()).ExecuteTest() THEN
	Expected		   := FALSE;
	DigitalInput.Force := E_ForceState.ForceOn;
	ForceVisitor.Force := E_ForceState.ForceOff;
	DigitalInput.Accept(ForceVisitor);
	Input  := TRUE;
	Actual := DigitalInput.IsActive;
	TestSuite.Test(__POUNAME()).AssertEqual(Expected, Actual);
END_IF
END_METHOD

METHOD ForceOnVisitor_NC
VAR
	Expected	 : BOOL;
	Actual		 : BOOL;
	Input		 : BOOL;
	DigitalInput : DigitalInput_NC('DigitalInput', Input);
	ForceVisitor : ForceVisitor;
END_VAR
IF TestSuite.Test(__POUNAME()).ExecuteTest() THEN
	Expected		   := TRUE;
	DigitalInput.Force := E_ForceState.ForceOff;
	ForceVisitor.Force := E_ForceState.ForceOn;
	DigitalInput.Accept(ForceVisitor);
	Input  := FALSE;
	Actual := DigitalInput.IsActive;
	TestSuite.Test(__POUNAME()).AssertEqual(Expected, Actual);
END_IF
END_METHOD

METHOD ForceOnVisitor_NO
VAR
	Expected	 : BOOL;
	Actual		 : BOOL;
	Input		 : BOOL;
	DigitalInput : DigitalInput_NO('DigitalInput', Input);
	ForceVisitor : ForceVisitor;
END_VAR
IF TestSuite.Test(__POUNAME()).ExecuteTest() THEN
	Expected		   := TRUE;
	DigitalInput.Force := E_ForceState.ForceOff;
	ForceVisitor.Force := E_ForceState.ForceOn;
	DigitalInput.Accept(ForceVisitor);
	Input  := FALSE;
	Actual := DigitalInput.IsActive;
	TestSuite.Test(__POUNAME()).AssertEqual(Expected, Actual);
END_IF
END_METHOD

METHOD UnforcedVisitor_NC
VAR
	Expected	 : BOOL;
	Actual		 : BOOL;
	Input		 : BOOL;
	DigitalInput : DigitalInput_NC('DigitalInput', Input);
	ForceVisitor : ForceVisitor;
END_VAR
IF TestSuite.Test(__POUNAME()).ExecuteTest() THEN
	Expected		   := TRUE;
	DigitalInput.Force := E_ForceState.ForceOn;
	ForceVisitor.Force := E_ForceState.Unforced;
	DigitalInput.Accept(ForceVisitor);
	Input  := FALSE;
	Actual := DigitalInput.IsActive;
	TestSuite.Test(__POUNAME()).AssertEqual(Expected, Actual);
END_IF
END_METHOD

METHOD UnforcedVisitor_NO
VAR
	Expected	 : BOOL;
	Actual		 : BOOL;
	Input		 : BOOL;
	DigitalInput : DigitalInput_NO('DigitalInput', Input);
	ForceVisitor : ForceVisitor;
END_VAR
IF TestSuite.Test(__POUNAME()).ExecuteTest() THEN
	Expected		   := FALSE;
	DigitalInput.Force := E_ForceState.ForceOn;
	ForceVisitor.Force := E_ForceState.Unforced;
	DigitalInput.Accept(ForceVisitor);
	Input  := FALSE;
	Actual := DigitalInput.IsActive;
	TestSuite.Test(__POUNAME()).AssertEqual(Expected, Actual);
END_IF
END_METHOD

END_FUNCTION_BLOCK

// ---- UnitTests/Recipe/Recipe_TEST.TcPOU
FUNCTION_BLOCK Recipe_TEST
VAR
	ActiveRecipe	: ST_Recipe;
	UpdateRecipe	: ST_Recipe;
	RecipeManagment : RecipeManagment('Test Recipe Mgmt', nRecipe := SIZEOF(ST_Recipe), pActiveRecipeData := ADR(ActiveRecipe), pUpdateRecipeData := ADR(UpdateRecipe));
END_VAR

FirstCycleLoadNoChange();
DetectChangesLReal();
UpdateChangesLReal();
DetectChangesDint();
UpdateChangesDint();
DetectChangesBool();
UpdateChangesBool();
AutoLoad();

METHOD AutoLoad
VAR
	Expected : BOOL;
	Actual	 : BOOL;
END_VAR
IF TestSuite.Test(__POUNAME()).ExecuteTest() THEN
	Expected								:= TRUE;
	UpdateRecipe.ValueA						:= 0.756;
	RecipeManagment.AutoLoadChangesToActive := TRUE;
	RecipeManagment.CyclicLogic();
	Actual := NOT RecipeManagment.ChangesPending AND ActiveRecipe.ValueA = 0.756;
	TestSuite.Test(__POUNAME()).AssertEqual(Expected, Actual);
END_IF
END_METHOD

METHOD DetectChangesBool
VAR
	Expected : BOOL;
	Actual	 : BOOL;
END_VAR
IF TestSuite.Test(__POUNAME()).ExecuteTest() THEN
	Expected			:= TRUE;
	UpdateRecipe.ValueC := TRUE;
	RecipeManagment.CyclicLogic();
	Actual := RecipeManagment.ChangesPending;
	TestSuite.Test(__POUNAME()).AssertEqual(Expected, Actual);
END_IF
END_METHOD

METHOD DetectChangesDint
VAR
	Expected : BOOL;
	Actual	 : BOOL;
END_VAR
IF TestSuite.Test(__POUNAME()).ExecuteTest() THEN
	Expected			:= TRUE;
	UpdateRecipe.ValueB := 584;
	RecipeManagment.CyclicLogic();
	Actual := RecipeManagment.ChangesPending;
	TestSuite.Test(__POUNAME()).AssertEqual(Expected, Actual);
END_IF
END_METHOD

METHOD DetectChangesLReal
VAR
	Expected : BOOL;
	Actual	 : BOOL;
END_VAR
IF TestSuite.Test(__POUNAME()).ExecuteTest() THEN
	Expected			:= TRUE;
	UpdateRecipe.ValueA := 0.0584;
	RecipeManagment.CyclicLogic();
	Actual := RecipeManagment.ChangesPending;
	TestSuite.Test(__POUNAME()).AssertEqual(Expected, Actual);
END_IF
END_METHOD

METHOD FirstCycleLoadNoChange
VAR
	Expected : BOOL;
	Actual	 : BOOL;
END_VAR
IF TestSuite.Test(__POUNAME()).ExecuteTest() THEN
	Expected := FALSE;
	RecipeManagment.CyclicLogic();
	Actual := RecipeManagment.ChangesPending;
	TestSuite.Test(__POUNAME()).AssertEqual(Expected, Actual);
END_IF
END_METHOD

METHOD UpdateChangesBool
VAR
	Expected : BOOL;
	Actual	 : BOOL;
END_VAR
IF TestSuite.Test(__POUNAME()).ExecuteTest() THEN
	Expected := TRUE;
	RecipeManagment.LoadChangesToActive();
	RecipeManagment.CyclicLogic();
	Actual := NOT RecipeManagment.ChangesPending AND ActiveRecipe.ValueC;
	TestSuite.Test(__POUNAME()).AssertEqual(Expected, Actual);
END_IF
END_METHOD

METHOD UpdateChangesDint
VAR
	Expected : BOOL;
	Actual	 : BOOL;
END_VAR
IF TestSuite.Test(__POUNAME()).ExecuteTest() THEN
	Expected := TRUE;
	RecipeManagment.LoadChangesToActive();
	RecipeManagment.CyclicLogic();
	Actual := NOT RecipeManagment.ChangesPending AND ActiveRecipe.ValueB = 584;
	TestSuite.Test(__POUNAME()).AssertEqual(Expected, Actual);
END_IF
END_METHOD

METHOD UpdateChangesLReal
VAR
	Expected : BOOL;
	Actual	 : BOOL;
END_VAR
IF TestSuite.Test(__POUNAME()).ExecuteTest() THEN
	Expected := TRUE;
	RecipeManagment.LoadChangesToActive();
	RecipeManagment.CyclicLogic();
	Actual := NOT RecipeManagment.ChangesPending AND ActiveRecipe.ValueA = 0.0584;
	TestSuite.Test(__POUNAME()).AssertEqual(Expected, Actual);
END_IF
END_METHOD

END_FUNCTION_BLOCK

// ---- UnitTests/Analog/Analog_TEST.TcPOU
FUNCTION_BLOCK Analog_TEST
VAR
END_VAR

AnalogInputReturnsCorrectValue();
AnalogInputReturnsRawValueCorrectly();
AnalogOutputGenericCheckValue();
AnalogOutputGenericCheckRawValue();
AnalogAcceptsForceOff();
AnalogAcceptsForceOn();
AnalogAcceptsForceValue();
AnalogGenericPassesDataInValidCorrectly();
AnalogGenericPassesDataValidCorrectly();
AnalogGenericPassesErrorCorrectly();
AnalogGenericPassesOverrangeCorrectly();
AnalogGenericPassesUnderrangeCorrectly();

METHOD AnalogAcceptsForceOff
VAR
	InputGeneric		 : INT;
	AnalogInput_Generic	 : AnalogInput('Input Generic', InputGeneric);
	Expected : INT;
	Actual	 : INT;
END_VAR
IF TestSuite.Test(__POUNAME()).ExecuteTest() THEN
	Expected								   := 0;
	InputGeneric := 750;
	AnalogInput_Generic.ForceValue := 300;
	AnalogInput_Generic.Force := E_ForceState.ForceOff;
	Actual							:= AnalogInput_Generic.RawValue;
	TestSuite.Test(__POUNAME()).AssertEqual(Expected, Actual);
END_IF
END_METHOD

METHOD AnalogAcceptsForceOn
VAR
	InputGeneric		 : INT;
	AnalogInput_Generic	 : AnalogInput('Input Generic', InputGeneric);
	Expected : INT;
	Actual	 : INT;
END_VAR
IF TestSuite.Test(__POUNAME()).ExecuteTest() THEN
	Expected								   := 425;
	InputGeneric := 750;
	AnalogInput_Generic.ForceValue := Expected;
	AnalogInput_Generic.Force := E_ForceState.ForceOn;
	Actual							:= AnalogInput_Generic.RawValue;
	TestSuite.Test(__POUNAME()).AssertEqual(Expected, Actual);
END_IF
END_METHOD

METHOD AnalogAcceptsForceValue
VAR
	InputGeneric		 : INT;
	AnalogInput_Generic	 : AnalogInput('Input Generic', InputGeneric);
	Expected : INT;
	Actual	 : INT;
END_VAR
IF TestSuite.Test(__POUNAME()).ExecuteTest() THEN
	Expected								   := 750;
	AnalogInput_Generic.ForceValue := Expected;
	Actual							:= AnalogInput_Generic.ForceValue;
	TestSuite.Test(__POUNAME()).AssertEqual(Expected, Actual);
END_IF
END_METHOD

METHOD AnalogGenericPassesDataInValidCorrectly
VAR
	InputGeneric		 : INT;
	AnalogStatus : ST_AnalogInputStatus_Generic;
	AnalogInput_Generic	 : AnalogInput_Generic('Input Generic', InputGeneric, AnalogStatus );

	Expected : BOOL := TRUE;
	Actual	 : BOOL;
END_VAR
IF TestSuite.Test(__POUNAME()).ExecuteTest() THEN
	AnalogStatus.WcState := 0;
	Actual									   := AnalogInput_Generic.DataValid	;
	TestSuite.Test(__POUNAME()).AssertEqual(Expected, Actual);
END_IF
END_METHOD

METHOD AnalogGenericPassesDataValidCorrectly
VAR
	InputGeneric		 : INT;
	AnalogStatus : ST_AnalogInputStatus_Generic;
	AnalogInput_Generic	 : AnalogInput_Generic('Input Generic', InputGeneric, AnalogStatus );

	Expected : BOOL := FALSE;
	Actual	 : BOOL;
END_VAR
IF TestSuite.Test(__POUNAME()).ExecuteTest() THEN
	AnalogStatus.WcState := 1;
	Actual									   := AnalogInput_Generic.DataValid	;
	TestSuite.Test(__POUNAME()).AssertEqual(Expected, Actual);
END_IF
END_METHOD

METHOD AnalogGenericPassesErrorCorrectly
VAR
	InputGeneric		 : INT;
	AnalogStatus : ST_AnalogInputStatus_Generic;
	AnalogInput_Generic	 : AnalogInput_Generic('Input Generic', InputGeneric, AnalogStatus );

	Expected : BOOL := TRUE;
	Actual	 : BOOL;
END_VAR
IF TestSuite.Test(__POUNAME()).ExecuteTest() THEN
	AnalogStatus.Error := 1;
	Actual									   := AnalogInput_Generic.Error	;
	TestSuite.Test(__POUNAME()).AssertEqual(Expected, Actual);
END_IF
END_METHOD

METHOD AnalogGenericPassesOverrangeCorrectly
VAR
	InputGeneric		 : INT;
	AnalogStatus : ST_AnalogInputStatus_Generic;
	AnalogInput_Generic	 : AnalogInput_Generic('Input Generic', InputGeneric, AnalogStatus );

	Expected : BOOL := TRUE;
	Actual	 : BOOL;
END_VAR
IF TestSuite.Test(__POUNAME()).ExecuteTest() THEN
	AnalogStatus.Overrange := 1;
	Actual									   := AnalogInput_Generic.Overrange	;
	TestSuite.Test(__POUNAME()).AssertEqual(Expected, Actual);
END_IF
END_METHOD

METHOD AnalogGenericPassesUnderrangeCorrectly
VAR
	InputGeneric		 : INT;
	AnalogStatus : ST_AnalogInputStatus_Generic;
	AnalogInput_Generic	 : AnalogInput_Generic('Input Generic', InputGeneric, AnalogStatus );

	Expected : BOOL := TRUE;
	Actual	 : BOOL;
END_VAR
IF TestSuite.Test(__POUNAME()).ExecuteTest() THEN
	AnalogStatus.Underrrange := 1;
	Actual									   := AnalogInput_Generic.Underrange	;
	TestSuite.Test(__POUNAME()).AssertEqual(Expected, Actual);
END_IF
END_METHOD

METHOD AnalogInputReturnsCorrectValue
VAR
	InputGeneric		 : INT;
	AnalogInput_Generic	 : AnalogInput('Input Generic', InputGeneric);

	Expected : LREAL;
	Actual	 : LREAL;
END_VAR
IF TestSuite.Test(__POUNAME()).ExecuteTest() THEN
	InputGeneric							   := 8192;
	Expected								   := 6.00015;
	AnalogInput_Generic.Scale.InputMaximum	   := 32767;
	AnalogInput_Generic.Scale.InputMinimum	   := 0.0;
	AnalogInput_Generic.Scale.OutputMaximum	   := 10;
	AnalogInput_Generic.Scale.OutputMinimum	   := 0.0;
	AnalogInput_Generic.CalibrateLinear.Gain   := 2;
	AnalogInput_Generic.CalibrateLinear.Offset := 1;
	Actual									   := floor(AnalogInput_Generic.Value * 100000) / 100000;
	TestSuite.Test(__POUNAME()).AssertEqual(Expected, Actual);
END_IF
END_METHOD

METHOD AnalogInputReturnsRawValueCorrectly
VAR
	InputGeneric		 : INT;
	AnalogInput_Generic	 : AnalogInput('Input', InputGeneric);

	Expected : LREAL;
	Actual	 : LREAL;
END_VAR
IF TestSuite.Test(__POUNAME()).ExecuteTest() THEN
	InputGeneric							   := 750;
	Expected								   := 750;

	Actual									   := AnalogInput_Generic.RawValue;
	TestSuite.Test(__POUNAME()).AssertEqual(Expected, Actual);
END_IF
END_METHOD

METHOD AnalogOutputGenericCheckRawValue
VAR
	Expected : LREAL;
	Actual	 : LREAL;
	OutputGeneric		 : INT;
	AnalogOutput_Generic : AnalogOutput('Output Generic', OutputGeneric);
END_VAR
IF TestSuite.Test(__POUNAME()).ExecuteTest() THEN
	AnalogOutput_Generic.RawValue				:= 750;
	Expected									:= 750;
	AnalogOutput_Generic.Scale.InputMaximum		:= 10; // Process Value from plc e.g. liters
	AnalogOutput_Generic.Scale.InputMinimum		:= -10;
	AnalogOutput_Generic.Scale.OutputMaximum	:= 1000; // Output to terminal
	AnalogOutput_Generic.Scale.OutputMinimum	:= -1000;
	AnalogOutput_Generic.CalibrateLinear.Gain	:= 2;
	AnalogOutput_Generic.CalibrateLinear.Offset := 1;
	Actual										:= AnalogOutput_Generic.RawValue;
	TestSuite.Test(__POUNAME()).AssertEqual(Expected, Actual);
END_IF
END_METHOD

METHOD AnalogOutputGenericCheckValue
VAR
	Expected : LREAL;
	Actual	 : LREAL;
	OutputGeneric		 : INT;
	AnalogOutput_Generic : AnalogOutput('Output Generic', OutputGeneric);
END_VAR
IF TestSuite.Test(__POUNAME()).ExecuteTest() THEN
	Expected									:= 750;
	AnalogOutput_Generic.Scale.InputMaximum		:= 10; // Process Value from plc e.g. liters
	AnalogOutput_Generic.Scale.InputMinimum		:= -10;
	AnalogOutput_Generic.Scale.OutputMaximum	:= 1000; // Output to terminal
	AnalogOutput_Generic.Scale.OutputMinimum	:= -1000;
	AnalogOutput_Generic.CalibrateLinear.Gain	:= 1;
	AnalogOutput_Generic.CalibrateLinear.Offset := 0;
	AnalogOutput_Generic.Value					:= 7.5;
	Actual										:= AnalogOutput_Generic.RawValue;
	TestSuite.Test(__POUNAME()).AssertEqual(Expected, Actual);
END_IF
END_METHOD

END_FUNCTION_BLOCK

// ---- UnitTests/Serial/SerialConnection_Tests.TcPOU
FUNCTION_BLOCK SerialConnection_Tests
VAR
END_VAR

ByteConnectionAcceptsSendByte_Test();
StringConnectionAcceptsSendString_Test();
ByteConnectionRejectsSendByteWithNoLineCtrl_Test();
StringConnectionRejectsSendStringWithNoLineCtrl_Test();
ByteConnectionAcceptsSerialLineSet_Test();
ByteConnectionRejectsNulSerialLineSet_Test();
StringConnectionAcceptsSerialLineSet_Test();
StringConnectionRejectsNulSerialLineSet_Test();
ByteConnectionFlagsRecievedByte_Test();
ByteConnectionRecievesByteCorrectly_Test();
StringConnectionFlagsRecievedString_Test();
StringConnectionRecievesStringCorrectly_Test();
ByteConnectionRejectsResetWithNoLineCtrl_Test();
ByteConnectionResetsRxCommBuffer_Test();
StringConnectionRejectsResetWithNoLineCtrl_Test();
StringConnectionResetsRxCommBuffer_Test();

METHOD ByteConnectionAcceptsSendByte_Test : BOOL
VAR
	Expected : BOOL := TRUE;
	Actual	 : BOOL;
	seriallineCtrl : SerialLineControl_ADS;
	serialConnection : SerialByteConnection(Name := 'Channel 1',SerialLineController := seriallineCtrl);
END_VAR
IF TestSuite.Test(__POUNAME()).ExecuteTest() THEN
	Actual := SUCCEEDED(serialConnection.SendAByte(1));
	TestSuite.Test(__POUNAME()).AssertEqual(Expected, Actual);
END_IF
END_METHOD

METHOD ByteConnectionAcceptsSerialLineSet_Test : BOOL
VAR
	Expected : BOOL := TRUE;
	Actual	 : BOOL;
	seriallineCtrl : SerialLineControl_ADS;
	serialConnection : SerialByteConnection(Name := 'Channel 1',SerialLineController := 0);
END_VAR
IF TestSuite.Test(__POUNAME()).ExecuteTest() THEN
	Actual := serialConnection.SetDependencies(seriallineCtrl);
	TestSuite.Test(__POUNAME()).AssertEqual(Expected, Actual);
END_IF
END_METHOD

METHOD ByteConnectionFlagsRecievedByte_Test : BOOL
VAR
	Expected : BOOL := TRUE;
	Actual	 : BOOL;
	seriallineCtrl : MockSerialLineCtrl;
	serialConnection : SerialByteConnection(Name := 'Channel 1',SerialLineController := seriallineCtrl);
END_VAR
IF TestSuite.Test(__POUNAME()).ExecuteTest() THEN
	seriallineCtrl.SetComBufferByte(4);
	serialConnection.CyclicLogic();
	serialConnection.CyclicLogic();
	Actual := serialConnection.ByteDataRecieved;
	TestSuite.Test(__POUNAME()).AssertEqual(Expected, Actual);
END_IF
END_METHOD

METHOD ByteConnectionRecievesByteCorrectly_Test : BOOL
VAR
	Expected : BOOL := TRUE;
	Actual	 : BOOL;
	seriallineCtrl : MockSerialLineCtrl;
	serialConnection : SerialByteConnection(Name := 'Channel 1',SerialLineController := seriallineCtrl);
	TestByte : BYTE := 4;
END_VAR
IF TestSuite.Test(__POUNAME()).ExecuteTest() THEN
	seriallineCtrl.SetComBufferByte(TestByte);
	serialConnection.CyclicLogic();
	serialConnection.CyclicLogic();
	IF serialConnection.ByteDataRecieved THEN
		Actual := serialConnection.ByteData = TestByte;
	END_IF
	TestSuite.Test(__POUNAME()).AssertEqual(Expected, Actual);
END_IF
END_METHOD

METHOD ByteConnectionRejectsNulSerialLineSet_Test
VAR
	Expected : BOOL := FALSE;
	Actual	 : BOOL;
	serialConnection : SerialByteConnection(Name := 'Channel 1',SerialLineController := 0);
END_VAR
IF TestSuite.Test(__POUNAME()).ExecuteTest() THEN
	Actual := serialConnection.SetDependencies(0);
	TestSuite.Test(__POUNAME()).AssertEqual(Expected, Actual);
END_IF
END_METHOD

METHOD ByteConnectionRejectsResetWithNoLineCtrl_Test : BOOL
VAR
	Expected : BOOL := TRUE;
	Actual	 : BOOL;
	serialConnection : SerialByteConnection(Name := 'Channel 1',SerialLineController := 0);
END_VAR
IF TestSuite.Test(__POUNAME()).ExecuteTest() THEN
	Actual := FAILED(serialConnection.Reset());
	TestSuite.Test(__POUNAME()).AssertEqual(Expected, Actual);
END_IF
END_METHOD

METHOD ByteConnectionRejectsSendByteWithNoLineCtrl_Test : BOOL
VAR
	Expected : BOOL := TRUE;
	Actual	 : BOOL;
	serialConnection : SerialByteConnection(Name := 'Channel 1',SerialLineController := 0);
END_VAR
IF TestSuite.Test(__POUNAME()).ExecuteTest() THEN
	Actual := FAILED(serialConnection.SendAByte(1));
	TestSuite.Test(__POUNAME()).AssertEqual(Expected, Actual);
END_IF
END_METHOD

METHOD ByteConnectionResetsRxCommBuffer_Test : BOOL
VAR
	Expected : BOOL := TRUE;
	Actual	 : BOOL;
	seriallineCtrl : MockSerialLineCtrl;
	serialConnection : SerialByteConnection(Name := 'Channel 1',SerialLineController := seriallineCtrl);
END_VAR
IF TestSuite.Test(__POUNAME()).ExecuteTest() THEN
	seriallineCtrl.SetComBufferByte(4);
	serialConnection.CyclicLogic();
	serialConnection.CyclicLogic();
	serialConnection.Reset();
	Actual := seriallineCtrl.rxBuffer.RdIdx = 0;
	TestSuite.Test(__POUNAME()).AssertEqual(Expected, Actual);
END_IF
END_METHOD

METHOD StringConnectionAcceptsSendString_Test : BOOL
VAR
	Expected : BOOL := TRUE;
	Actual	 : BOOL;
	seriallineCtrl : SerialLineControl_ADS;
	serialConnection : SerialStringConnection(Name := 'Channel 1',SerialLineController := seriallineCtrl);
END_VAR
IF TestSuite.Test(__POUNAME()).ExecuteTest() THEN
	Actual := SUCCEEDED(serialConnection.SendAString('Bob'));
	TestSuite.Test(__POUNAME()).AssertEqual(Expected, Actual);
END_IF
END_METHOD

METHOD StringConnectionAcceptsSerialLineSet_Test : BOOL
VAR
	Expected : BOOL := TRUE;
	Actual	 : BOOL;
	seriallineCtrl : SerialLineControl_ADS;
	serialConnection : SerialStringConnection(Name := 'Channel 1',SerialLineController := 0);
END_VAR
IF TestSuite.Test(__POUNAME()).ExecuteTest() THEN
	Actual := serialConnection.SetDependencies(seriallineCtrl);
	TestSuite.Test(__POUNAME()).AssertEqual(Expected, Actual);
END_IF
END_METHOD

METHOD StringConnectionFlagsRecievedString_Test : BOOL
VAR
	Expected : BOOL := TRUE;
	Actual	 : BOOL;
	seriallineCtrl : MockSerialLineCtrl;
	serialConnection : SerialStringConnection(Name := 'Channel 1',SerialLineController := seriallineCtrl);
END_VAR
IF TestSuite.Test(__POUNAME()).ExecuteTest() THEN
	seriallineCtrl.SetComBufferString('$02 I Love Chips $03',20);
	serialConnection.SetSerialConfiguration('$02','$03');
	serialConnection.CyclicLogic();
	serialConnection.CyclicLogic();
	serialConnection.CyclicLogic();
	Actual := serialConnection.StringRecieved;
	TestSuite.Test(__POUNAME()).AssertEqual(Expected, Actual);
END_IF
END_METHOD

METHOD StringConnectionRecievesStringCorrectly_Test : BOOL
VAR
	Expected : BOOL := TRUE;
	Actual	 : BOOL;
	seriallineCtrl : MockSerialLineCtrl;
	serialConnection : SerialStringConnection(Name := 'Channel 1',SerialLineController := seriallineCtrl);
	testString : T_MaxString := '$02 I Love Chips $03';
END_VAR
IF TestSuite.Test(__POUNAME()).ExecuteTest() THEN
	seriallineCtrl.SetComBufferString('$02 I Love Chips $03',20);
	serialConnection.SetSerialConfiguration('$02','$03');
	serialConnection.CyclicLogic();
	serialConnection.CyclicLogic();
	serialConnection.CyclicLogic();
	IF serialConnection.StringRecieved THEN
		Actual := serialConnection.StringData = testString;
	END_IF
	TestSuite.Test(__POUNAME()).AssertEqual(Expected, Actual);
END_IF
END_METHOD

METHOD StringConnectionRejectsNulSerialLineSet_Test
VAR
	Expected : BOOL := FALSE;
	Actual	 : BOOL;
	serialConnection : SerialStringConnection(Name := 'Channel 1',SerialLineController := 0);
END_VAR
IF TestSuite.Test(__POUNAME()).ExecuteTest() THEN
	Actual := serialConnection.SetDependencies(0);
	TestSuite.Test(__POUNAME()).AssertEqual(Expected, Actual);
END_IF
END_METHOD

METHOD StringConnectionRejectsResetWithNoLineCtrl_Test : BOOL
VAR
	Expected : BOOL := TRUE;
	Actual	 : BOOL;
	serialConnection : SerialStringConnection(Name := 'Channel 1',SerialLineController := 0);
END_VAR
IF TestSuite.Test(__POUNAME()).ExecuteTest() THEN
	Actual := FAILED(serialConnection.Reset());
	TestSuite.Test(__POUNAME()).AssertEqual(Expected, Actual);
END_IF
END_METHOD

METHOD StringConnectionRejectsSendStringWithNoLineCtrl_Test : BOOL
VAR
	Expected : BOOL := TRUE;
	Actual	 : BOOL;
	serialConnection : SerialStringConnection(Name := 'Channel 1',SerialLineController := 0);
END_VAR
IF TestSuite.Test(__POUNAME()).ExecuteTest() THEN
	Actual := FAILED(serialConnection.SendAString('Bob'));
	TestSuite.Test(__POUNAME()).AssertEqual(Expected, Actual);
END_IF
END_METHOD

METHOD StringConnectionResetsRxCommBuffer_Test : BOOL
VAR
	Expected : BOOL := TRUE;
	Actual	 : BOOL;
	seriallineCtrl : MockSerialLineCtrl;
	serialConnection : SerialStringConnection(Name := 'Channel 1',SerialLineController := seriallineCtrl);
END_VAR
IF TestSuite.Test(__POUNAME()).ExecuteTest() THEN
	seriallineCtrl.SetComBufferByte(4);
	serialConnection.CyclicLogic();
	serialConnection.CyclicLogic();
	serialConnection.Reset();
	Actual := seriallineCtrl.rxBuffer.RdIdx = 0;
	TestSuite.Test(__POUNAME()).AssertEqual(Expected, Actual);
END_IF
END_METHOD

END_FUNCTION_BLOCK

// ---- _Mockups/SerialLineCtrl/MockSerialLineCtrl.TcPOU
FUNCTION_BLOCK MockSerialLineCtrl EXTENDS SerialLineControl_ADS
VAR
END_VAR

METHOD SetComBufferByte
VAR_INPUT
	ByteValue : BYTE;
END_VAR
rxComBuffer.Buffer[0] := ByteValue;
rxComBuffer.RdIdx := 0;
rxComBuffer.WrIdx := 0;
rxComBuffer.Count := 1;
rxComBuffer.FreeByte := 301;
END_METHOD

METHOD SetComBufferString
VAR_INPUT
	TestString : T_MaxString;
	StringSize : UINT;
END_VAR
VAR
	InterimString : T_MaxString;
	ByteOutput: ARRAY [0..Tc2_Utilities.MAX_STRING_LENGTH] OF BYTE;
	i : UDINT;
END_VAR
ByteOutput := MAXSTRING_TO_BYTEARR(TestString);
FOR i := StringSize - 1 TO MAX_STRING_LENGTH DO
	ByteOutput[i] := 0;
END_FOR
FOR i := 0 TO MAX_STRING_LENGTH DO
	rxComBuffer.Buffer[i] := ByteOutput[i];
END_FOR
rxComBuffer.RdIdx := 0;
rxComBuffer.WrIdx := 0;
rxComBuffer.Count := StringSize;
rxComBuffer.FreeByte := 301;
END_METHOD

END_FUNCTION_BLOCK

// ---- UnitTests/Axis/Axis_Test.TcPOU
FUNCTION_BLOCK Axis_Test
VAR
	AxisRef		: Tc2_MC2.AXIS_REF;
	Axis		: Mc2AxisPTP('Unit Test Axis', AxisRef) := (Override := 100.0);
	StartupTime : TON;
END_VAR

Axis.CyclicLogic();
StartupTime(IN := TRUE, PT := T#1S);
IF NOT StartupTime.Q THEN
	RETURN;
END_IF

Initialize();
Enable();
JogForward();
JogBackward();
MoveAbsoluteToStop();
Stop();
MoveAbsoluteToPoint();
Home();
Disable();
Error();
Reset();

METHOD Disable
VAR_INST
	Expected  : BOOL;
	Actual	  : BOOL;
	DoneTimer : TON;
END_VAR
IF TestSuite.Test(__POUNAME()).ExecuteTest() THEN
	Expected := TRUE;
	DoneTimer(IN := TRUE, PT := T#50MS);
	Axis.Disable();
	IF DoneTimer.Q THEN
		Actual := NOT Axis.Enabled AND NOT Axis.Busy AND NOT Axis.Error;
		TestSuite.Test(__POUNAME()).AssertEqual(Expected, Actual);
	END_IF
END_IF
END_METHOD

METHOD Enable
VAR_INST
	Expected  : BOOL;
	Actual	  : BOOL;
	DoneTimer : TON;
END_VAR
IF TestSuite.Test(__POUNAME()).ExecuteTest() THEN
	Expected := TRUE;
	DoneTimer(IN := TRUE, PT := T#50MS);
	Axis.Enable();
	IF DoneTimer.Q THEN
		Actual := Axis.Enabled AND NOT Axis.Busy AND NOT Axis.Error;
		TestSuite.Test(__POUNAME()).AssertEqual(Expected, Actual);
	END_IF
END_IF
END_METHOD

METHOD Error
VAR_INST
	Expected  : BOOL;
	Actual	  : BOOL;
	DoneTimer : TON;
END_VAR
IF TestSuite.Test(__POUNAME()).ExecuteTest() THEN
	Expected := TRUE;
	DoneTimer(IN := TRUE, PT := T#50MS);
	Axis.MoveAbsolute(20);
	IF DoneTimer.Q THEN
		Actual := (Axis.ErrorId <> 0) AND NOT Axis.Busy AND Axis.Error;
		TestSuite.Test(__POUNAME()).AssertEqual(Expected, Actual);
	END_IF
END_IF
END_METHOD

METHOD Home
VAR_INST
	Expected  : BOOL;
	Actual	  : BOOL;
	DoneTimer : TON;
	Command	  : BOOL := TRUE;
END_VAR
IF TestSuite.Test(__POUNAME()).ExecuteTest() THEN
	Expected := TRUE;
	DoneTimer(IN := TRUE, PT := T#100MS);
	IF Command AND NOT Axis.Busy THEN
		Command := FALSE;
		Axis.Home();
	END_IF

	IF DoneTimer.Q THEN
		Actual := CompareLREAL(Axis.ActualVelocity, 0, 0.1) AND CompareLREAL(Axis.ActualPosition, 0, 0.1) AND NOT Axis.Busy AND NOT Axis.Error;
		TestSuite.Test(__POUNAME()).AssertEqual(Expected, Actual);
	END_IF
END_IF
END_METHOD

METHOD Initialize
VAR_INST
	Expected  : BOOL;
	Actual	  : BOOL;
	DoneTimer : TON;
END_VAR
IF TestSuite.Test(__POUNAME()).ExecuteTest() THEN
	DoneTimer(IN := TRUE, PT := T#250MS);
	Expected := TRUE;
	IF DoneTimer.Q THEN
		Actual := Axis.Initialized AND NOT Axis.Error;
		TestSuite.Test(__POUNAME()).AssertEqual(Expected, Actual);
	END_IF
END_IF
END_METHOD

METHOD JogBackward
VAR_INST
	Expected  : BOOL;
	Actual	  : BOOL;
	DoneTimer : TON;
END_VAR
IF TestSuite.Test(__POUNAME()).ExecuteTest() THEN
	Expected := TRUE;
	DoneTimer(IN := TRUE, PT := T#1S);
	Axis.Jog(FALSE, TRUE);
	IF DoneTimer.Q THEN
		Actual := (Axis.ActualVelocity < 0) AND Axis.Busy AND NOT Axis.Error;
		TestSuite.Test(__POUNAME()).AssertEqual(Expected, Actual);
		Axis.Jog(FALSE, FALSE);
	END_IF
END_IF
END_METHOD

METHOD JogForward
VAR_INST
	Expected  : BOOL;
	Actual	  : BOOL;
	DoneTimer : TON;
END_VAR
IF TestSuite.Test(__POUNAME()).ExecuteTest() THEN
	Expected := TRUE;
	DoneTimer(IN := TRUE, PT := T#100MS);
	Axis.Jog(TRUE, FALSE);
	IF DoneTimer.Q THEN
		Actual := (Axis.ActualVelocity > 0) AND Axis.Busy AND NOT Axis.Error;
		TestSuite.Test(__POUNAME()).AssertEqual(Expected, Actual);
		Axis.Jog(FALSE, FALSE);
	END_IF
END_IF
END_METHOD

METHOD MoveAbsoluteToPoint
VAR_INST
	Expected  : BOOL;
	Actual	  : BOOL;
	DoneTimer : TON;
	Command	  : BOOL := TRUE;
END_VAR
IF TestSuite.Test(__POUNAME()).ExecuteTest() THEN
	Expected := TRUE;
	DoneTimer(IN := TRUE, PT := T#2S);
	IF Command AND NOT Axis.Busy THEN
		Command := FALSE;
		Axis.MoveAbsolute(100);
	END_IF

	IF DoneTimer.Q THEN
		Actual := CompareLREAL(Axis.ActualVelocity, 0, 0.1) AND CompareLREAL(Axis.ActualPosition, 100, 0.1) AND NOT Axis.Busy AND NOT Axis.Error;
		TestSuite.Test(__POUNAME()).AssertEqual(Expected, Actual);
	END_IF
END_IF
END_METHOD

METHOD MoveAbsoluteToStop
VAR_INST
	Expected  : BOOL;
	Actual	  : BOOL;
	DoneTimer : TON;
	Command	  : BOOL := TRUE;
END_VAR
IF TestSuite.Test(__POUNAME()).ExecuteTest() THEN
	Expected := TRUE;
	DoneTimer(IN := TRUE, PT := T#1S);
	IF Command AND NOT Axis.Busy THEN
		Command := FALSE;
		Axis.MoveAbsolute(1000);
	END_IF

	IF DoneTimer.Q THEN
		Actual := (Axis.ActualVelocity > 0) AND Axis.Busy AND NOT Axis.Error;
		TestSuite.Test(__POUNAME()).AssertEqual(Expected, Actual);
	END_IF
END_IF
END_METHOD

METHOD Reset
VAR_INST
	Expected  : BOOL;
	Actual	  : BOOL;
	DoneTimer : TON;
	Command	  : BOOL := TRUE;
END_VAR
IF TestSuite.Test(__POUNAME()).ExecuteTest() THEN
	Expected := TRUE;
	DoneTimer(IN := TRUE, PT := T#500MS);
	IF Command THEN
		Command := FALSE;
		Axis.Reset();
	END_IF

	IF DoneTimer.Q THEN
		Actual := (Axis.ErrorId = 0) AND NOT Axis.Busy AND NOT Axis.Error;
		TestSuite.Test(__POUNAME()).AssertEqual(Expected, Actual);
	END_IF
END_IF
END_METHOD

METHOD Stop
VAR_INST
	Expected  : BOOL;
	Actual	  : BOOL;
	DoneTimer : TON;
END_VAR
IF TestSuite.Test(__POUNAME()).ExecuteTest() THEN
	Expected := TRUE;
	DoneTimer(IN := TRUE, PT := T#500MS);
	Axis.Stop();
	IF DoneTimer.Q THEN
		Actual := CompareLREAL(Axis.ActualVelocity, 0, 0.1) AND NOT Axis.Busy AND NOT Axis.Error;
		TestSuite.Test(__POUNAME()).AssertEqual(Expected, Actual);
	END_IF
END_IF
END_METHOD

END_FUNCTION_BLOCK

// ---- UnitTests/EtherCat/EtherCatMaster_TEST.TcPOU
FUNCTION_BLOCK EtherCatMaster_TEST
VAR
	Provider : EtherCatEventProvider_Mockup('EtherCAT Event Provider');
	Master	 : EtherCatMaster_Mockup('EtherCAT Master Mock', EcStartupCycles := 1);
	Device	 : EtherCatIoDevice('Io Device');
	State	 : ST_EcExtendedSlaveState;
	Config	 : ST_EcSlaveConfigData;
END_VAR

IoDeviceStateFlags();
IoDeviceDiagnosticFlags();
IoDeviceCoeNullWithoutMailbox();
IoDeviceCoeWithMailbox();
MasterEventOncePerDevStateChange();
SlaveIndexByAddress();
SlaveIndexByAddressOutsideDenseRange();
SlaveRegistryNameAndHotConnect();
IoDeviceByAddrUsesMap();
AdsFailureKeepsErrorId();

// A failing slave state read aborts the sequence with ErrorSource Ads and the error id of the
// function block (or 16#745 on watchdog), never the former placeholder 999.
METHOD AdsFailureKeepsErrorId
VAR_INST
	Expected : BOOL;
	Actual	 : BOOL;
	Seq		 : UDINT;
	Cycles	 : UDINT;
END_VAR
IF TestSuite.Test(__POUNAME()).ExecuteTest() THEN
	Expected := TRUE;
	CASE Seq OF
		0:
			Master.LoadConfiguration(10);
			Master.SetMasterAmsNetId('1.2.3.4.5.6'); // no route: the read fails or times out
			Master.StartDiagnostic();
			Seq := 10;

		10:
			Master.RunSlaveState();
			Cycles := Cycles + 1;
			IF NOT Master.Busy OR Cycles > 2000 THEN
				Seq := 20;
			END_IF

		20:
			Actual := Master.Error AND (Master.ErrorSource = E_EcErrorSource.Ads) AND (Master.ErrorId <> 999) AND (Master.ErrorId <> 0);
			TestSuite.Test(__POUNAME()).AssertEqual(Expected, Actual);
	END_CASE
END_IF
END_METHOD

// The device returned for an address reflects the state of exactly that configured slave.
METHOD IoDeviceByAddrUsesMap
VAR_INST
	Expected : BOOL;
	Actual	 : BOOL;
END_VAR
IF TestSuite.Test(__POUNAME()).ExecuteTest() THEN
	Expected := TRUE;
	Master.LoadConfiguration(10);
	Master.SetSlaveState(Index := 2, DeviceState := 16#04, LinkState := 16#00); // slave at 1003 in SAFEOP
	Actual := Master.GetIoDeviceByAddr(1003).SafeOp AND Master.GetIoDeviceByAddr(1002).OP AND Master.GetIoDeviceByAddr(1004).OP AND NOT Master.GetIoDeviceByAddr(2000).OP;
	TestSuite.Test(__POUNAME()).AssertEqual(Expected, Actual);
END_IF
END_METHOD

METHOD IoDeviceCoeNullWithoutMailbox
VAR_INST
	Expected : STRING;
	Actual	 : STRING;
END_VAR
IF TestSuite.Test(__POUNAME()).ExecuteTest() THEN
	Expected			 := 'Null Terminal';
	Config.nMailboxInSize := 0;
	Device.Configuration REF= Config;
	Actual				 := Device.CoE.Name;
	TestSuite.Test(__POUNAME()).AssertEqual(Expected, Actual);
END_IF
END_METHOD

METHOD IoDeviceCoeWithMailbox
VAR_INST
	Expected : STRING;
	Actual	 : STRING;
END_VAR
IF TestSuite.Test(__POUNAME()).ExecuteTest() THEN
	Expected			 := 'CoE Terminal';
	Config.nMailboxInSize := 128;
	Config.nAddr		 := 1001;
	Device.Configuration REF= Config;
	Actual				 := Device.CoE.Name;
	TestSuite.Test(__POUNAME()).AssertEqual(Expected, Actual);
END_IF
END_METHOD

// deviceState bits 4..7 (error, invalid VPRS, init command error, disabled) are flags on top of the ESM state.
METHOD IoDeviceDiagnosticFlags
VAR_INST
	Expected : BOOL;
	Actual	 : BOOL;
END_VAR
IF TestSuite.Test(__POUNAME()).ExecuteTest() THEN
	Expected		  := TRUE;
	Device.State	 REF= State;
	State.deviceState := 16#F8; // OP with all four diagnostic bits set
	State.linkState	  := 16#00;
	Actual			  := Device.OP AND Device.DeviceError AND Device.InvalidVPRS AND Device.InitCmdError AND Device.Disabled;
	TestSuite.Test(__POUNAME()).AssertEqual(Expected, Actual);
END_IF
END_METHOD

METHOD IoDeviceStateFlags
VAR_INST
	Expected : BOOL;
	Actual	 : BOOL;
END_VAR
IF TestSuite.Test(__POUNAME()).ExecuteTest() THEN
	Expected		  := TRUE;
	Device.State	 REF= State;
	State.deviceState := 16#04; // SAFEOP, no diagnostic bits
	State.linkState	  := 16#00;
	Actual			  := Device.SafeOp AND NOT Device.OP AND NOT Device.PreOp AND NOT Device.Init AND NOT Device.Bootstrap
						 AND NOT Device.DeviceError AND NOT Device.InvalidVPRS AND NOT Device.InitCmdError AND NOT Device.Disabled;
	TestSuite.Test(__POUNAME()).AssertEqual(Expected, Actual);
END_IF
END_METHOD

// The MasterError event is raised once per DevState change, not every cycle the state persists.
METHOD MasterEventOncePerDevStateChange
VAR_INST
	Expected : UINT;
	Actual	 : UINT;
END_VAR
IF TestSuite.Test(__POUNAME()).ExecuteTest() THEN
	Expected := 1;
	Master.LoadConfiguration(10);
	Master.RegisterEventProvider(Provider);
	Master.SetMasterDevState(DevState := 16#0001, SlaveCount := 9); // link error, one slave missing
	Master.RunMasterState();
	Master.RunMasterState();
	Master.RunMasterState();
	Actual := Provider.MasterEventCount;
	TestSuite.Test(__POUNAME()).AssertEqual(Expected, Actual);
END_IF
END_METHOD

METHOD SlaveIndexByAddress
VAR_INST
	Expected : DINT;
	Actual	 : DINT;
END_VAR
IF TestSuite.Test(__POUNAME()).ExecuteTest() THEN
	Expected := 4;
	Master.LoadConfiguration(10);
	Actual := Master.GetSlaveIndexByAddr(1005);
	TestSuite.Test(__POUNAME()).AssertEqual(Expected, Actual);
END_IF
END_METHOD

// A user assigned address outside 1001.. is found by the linear fallback; unknown addresses give -1.
METHOD SlaveIndexByAddressOutsideDenseRange
VAR_INST
	Expected : BOOL;
	Actual	 : BOOL;
END_VAR
IF TestSuite.Test(__POUNAME()).ExecuteTest() THEN
	Expected := TRUE;
	Master.LoadConfiguration(10);
	Master.SetSlaveAddress(Index := 7, Addr := 60000);
	Actual := (Master.GetSlaveIndexByAddr(60000) = 7) AND (Master.GetSlaveIndexByAddr(1008) = -1) AND (Master.GetSlaveIndexByAddr(999) = -1);
	TestSuite.Test(__POUNAME()).AssertEqual(Expected, Actual);
END_IF
END_METHOD

// The master serves SyncUnitTask through I_EcSlaveRegistry: name and hot connect flag by index,
// safe defaults outside the configured range.
METHOD SlaveRegistryNameAndHotConnect
VAR_INST
	Expected : BOOL;
	Actual	 : BOOL;
	Registry : I_EcSlaveRegistry;
END_VAR
IF TestSuite.Test(__POUNAME()).ExecuteTest() THEN
	Expected := TRUE;
	Master.LoadConfiguration(10);
	Master.SetHotConnect(Index := 3);
	Registry := Master;
	Actual	 := (Registry.ConfiguredSlaveCount = 10)
				AND (Registry.GetSlaveName(4) = 'Slave5')
				AND Registry.IsHotConnectMember(3)
				AND NOT Registry.IsHotConnectMember(4)
				AND (Registry.GetSlaveName(10) = '')
				AND NOT Registry.IsHotConnectMember(10);
	TestSuite.Test(__POUNAME()).AssertEqual(Expected, Actual);
END_IF
END_METHOD

END_FUNCTION_BLOCK

// ---- _Mockups/EtherCat/EtherCatEventProvider_Mockup.TcPOU
// Counts the diagnostic events an EtherCatMaster raises instead of publishing TcEvents.
FUNCTION_BLOCK EtherCatEventProvider_Mockup EXTENDS Component IMPLEMENTS I_EtherCatDiagnosticEventProvider
VAR
	_MasterEventCount	: UINT;
	_SyncUnitEventCount : UINT;
	_ResetCount			: UINT;
	_LastEventId		: UDINT;
	_LastArgument1		: STRING;
	_LastArgument2		: STRING;
END_VAR

METHOD GetHighestActiveEventReaction : DINT
GetHighestActiveEventReaction := 0;
END_METHOD

METHOD GetHighestActiveEventSeverity : TcEventSeverity
GetHighestActiveEventSeverity := TcEventSeverity.Verbose;
END_METHOD

PROPERTY LastArgument1 : STRING
GET
LastArgument1 := _LastArgument1;
END_GET
END_PROPERTY

PROPERTY LastArgument2 : STRING
GET
LastArgument2 := _LastArgument2;
END_GET
END_PROPERTY

PROPERTY LastEventId : UDINT
GET
LastEventId := _LastEventId;
END_GET
END_PROPERTY

// Number of RaiseEtherCatDiagnosticEvent calls (master and slave events).
PROPERTY MasterEventCount : UINT
GET
MasterEventCount := _MasterEventCount;
END_GET
END_PROPERTY

METHOD RaiseEtherCatDiagnosticEvent
VAR_INPUT
	EventId	  : UDINT;
	Argument1 : STRING := '';
	Argument2 : STRING := '';
	Argument3 : STRING := '';
END_VAR
_MasterEventCount := _MasterEventCount + 1;
_LastEventId	  := EventId;
_LastArgument1	  := Argument1;
_LastArgument2	  := Argument2;
END_METHOD

METHOD RaiseSyncUnitEvent
VAR_INPUT
	EventId	  : UDINT;
	Argument1 : STRING := '';
	Argument2 : STRING := '';
	Argument3 : STRING := '';
END_VAR
_SyncUnitEventCount := _SyncUnitEventCount + 1;
_LastEventId		:= EventId;
_LastArgument1		:= Argument1;
_LastArgument2		:= Argument2;
END_METHOD

METHOD Reset
_ResetCount := _ResetCount + 1;
END_METHOD

PROPERTY ResetCount : UINT
GET
ResetCount := _ResetCount;
END_GET
END_PROPERTY

METHOD SetEventReactions
VAR_INPUT
	Verbose	 : DINT := 0;
	Info	 : DINT := 1;
	Warning	 : DINT := 2;
	Error	 : DINT := 3;
	Critical : DINT := 4;
END_VAR
END_METHOD

PROPERTY SyncUnitEventCount : UINT
GET
SyncUnitEventCount := _SyncUnitEventCount;
END_GET
END_PROPERTY

END_FUNCTION_BLOCK

// ---- _Mockups/EtherCat/EtherCatMaster_Mockup.TcPOU
// EtherCatMaster with its hardware inputs and slave arrays fed from the test instead of the master
// device. Exposes the protected evaluation steps so they can be driven without ADS or an EtherCAT master.
FUNCTION_BLOCK EtherCatMaster_Mockup EXTENDS EtherCatMaster<1, 1>
VAR
END_VAR

// Same inputs as EtherCatMaster.FB_Init; the base constructor receives them implicitly.
METHOD FB_Init : BOOL
VAR_INPUT
	bInitRetains	: BOOL; // TRUE: the retain variables are initialized (reset warm / reset cold)
	bInCopyCode		: BOOL; // TRUE: the instance will be copied to the copy code afterward (online change)
	Name			: T_MaxString;
	EcStartupCycles : UINT;
END_VAR
END_METHOD

// Current step of the slave diagnostic sequence (0 = idle).
PROPERTY DiagnosticStep : UDINT
GET
DiagnosticStep := SlaveSequence;
END_GET
END_PROPERTY

// Fakes a finished Initialize: Count slaves named Slave1..SlaveN at addresses 1001.., all OP, no mailbox.
METHOD LoadConfiguration
VAR_INPUT
	Count : UINT;
END_VAR

VAR
	i : UINT;
	n : UINT;
END_VAR
n := MIN(Count, MAX_EC_SLAVES + 1);

EcMaster.CfgSlaveCount := n;
EcMaster.SlaveCount	   := n;
SlaveCountUsed		   := n;

i := 0;
WHILE i < n DO
	ConfiguredSlaveInfo[i].nAddr		  := FIRST_SLAVE_ADDR + i;
	ConfiguredSlaveInfo[i].sName		  := CONCAT('Slave', TO_STRING(i + 1));
	ConfiguredSlaveInfo[i].nMailboxInSize := 0;
	SlavesState[i].deviceState			  := 16#08; // OP
	SlavesState[i].linkState			  := 16#00;
	SlaveTopologyInfo[i].nStatusBits	  := 0;	// no hot connect group (see SetHotConnect)
	IoDevice[i].Name					  := ConfiguredSlaveInfo[i].sName;
	IoDevice[i].State					  REF= SlavesState[i];
	IoDevice[i].Configuration			  REF= ConfiguredSlaveInfo[i];
	i									  := i + 1;
END_WHILE

BuildAddrToIndex();
Initialized := TRUE;
END_METHOD

// One evaluation of the master DevState (normally done by CyclicLogic).
METHOD RunMasterState : BOOL
RunMasterState := MasterState();
END_METHOD

// One cycle of the slave diagnostic sequence (normally done by CyclicLogic).
METHOD RunSlaveState
SlaveState();
_Busy := SlaveSequence <> 0;
END_METHOD

// Target of the diagnostic ADS reads (normally taken from EcMaster.AmsNetID in Initialize).
METHOD SetMasterAmsNetId
VAR_INPUT
	NetId : T_AmsNetId;
END_VAR
_MasterAmsNetId := NetId;
END_METHOD

// Fakes the master process image: DevState word and number of slaves currently on the bus.
METHOD SetMasterDevState
VAR_INPUT
	DevState   : UINT;
	SlaveCount : UINT;
END_VAR
EcMaster.DevState	:= DevState;
EcMaster.SlaveCount := SlaveCount;
END_METHOD

// Gives the configured slave Index another EtherCAT address and rebuilds the address map.
METHOD SetSlaveAddress
VAR_INPUT
	Index : UINT;
	Addr  : UINT;
END_VAR
ConfiguredSlaveInfo[Index].nAddr := Addr;
BuildAddrToIndex();
END_METHOD

// Fakes the topology read: marks one slave as member of a hot connect group.
METHOD SetHotConnect
VAR_INPUT
	Index : UINT;
END_VAR
SlaveTopologyInfo[Index].nStatusBits.4 := TRUE;
END_METHOD

// Fakes the state read of one slave.
METHOD SetSlaveState
VAR_INPUT
	Index		: UINT;
	DeviceState : BYTE;
	LinkState	: BYTE;
END_VAR
SlavesState[Index].deviceState := DeviceState;
SlavesState[Index].linkState   := LinkState;
END_METHOD

// Requests a slave diagnostic sequence (normally triggered by ChangeCount, slave count or frame WC state).
METHOD StartDiagnostic
RunSlaveDiag := TRUE;
END_METHOD

END_FUNCTION_BLOCK

// ---- UnitTests/AnyBuffer/AnyBuffer_TEST.TcPOU
PROGRAM AnyBuffer_TEST

// TEST_AnyBuffer_Clear();
// TEST_AnyBuffer_DeleteAtIndex();
// TEST_AnyBuffer_PeekAtIndex();
// TEST_AnyBuffer_ReplaceAtIndex();
// TEST_AnyBuffer_PushLeft();
// TEST_AnyBuffer_PushRight();
// TEST_AnyBuffer_PopLeft();
// TEST_AnyBuffer_PopRight();
// TEST_AnyBuffer_PopAtIndex();
// TEST_AnyBuffer_InsertAtIndex();

END_PROGRAM

// ---- _Mockups/AnyBuffer/Samples_AnyBuffer.TcPOU
PROGRAM Samples_AnyBuffer
(*
## Recent Performance Optimizations - Summary of Changes

### 1. FifoBuffer Optimization
**Changed from inefficient to efficient FIFO implementation:**
- **Before**: Used `AppendLeft` (O(n) - shifts all elements) for Push and `PopRight` (O(1)) for Pop
- **After**: Uses `AppendRight` (O(1) - no shifting) for Push and `PopLeft` (O(n)) for Pop
- **Benefit**: Push operations are now constant-time, which is much more common than Pop in FIFO queues
- **Performance**: Push now O(1) instead of O(n)
- **Documentation**: Updated all documentation to reflect the new behavior and performance characteristics

### 2. RingBuffer - Eliminated All Shifting Operations
**Implemented proper circular buffer with head/tail pointers:**
- **Added tracking variables**: `headIndex`, `tailIndex`, `elementCount`
- **Push**: Now uses circular indexing to overwrite oldest element **without any shifting** (true O(1))
- **Pop**: Uses `PeekAtIndex` with circular head pointer advancement **without shifting** (O(1))
- **Before**: Used `PopLeft()` which shifted all elements (O(n) operation)
- **After**: Direct circular buffer implementation with no shifting at all
- **Performance**: Both Push and Pop are now true O(1) constant-time operations

### 3. New WriteAtIndex Method in AnyBuffer
**Added low-level method for direct buffer access:**
- **Purpose**: Write to any physical index (0 to capacity-1) without changing buffer counters
- **Key difference from ReplaceAtIndex**:
  - `ReplaceAtIndex`: Only writes to logical indices (requires elements to exist)
  - `WriteAtIndex`: Writes to physical indices (works on empty buffer)
- **Use case**: Perfect for circular buffer implementations that manage their own counters
- **Documentation**: Comprehensive documentation with warnings about low-level nature

### 4. RingBuffer Updated to Use WriteAtIndex
- **Replaced** `ReplaceAtIndex` with `WriteAtIndex` for both initial fill and overwrite
- **Benefit**: No longer requires buffer to have elements, RingBuffer manages its own `elementCount`
- **Documentation**: Updated all RingBuffer documentation to reflect use of WriteAtIndex

### Performance Improvements Summary

| Operation | Before | After |
|-----------|--------|-------|
| **FifoBuffer.Push** | O(n) - shifts all | O(1) - append right |
| **FifoBuffer.Pop** | O(1) - no shift | O(n) - shift left |
| **RingBuffer.Push** | O(n) - PopLeft shifts | O(1) - direct write |
| **RingBuffer.Pop** | O(n) - PopLeft shifts | O(1) - PeekAtIndex |

**Result**: RingBuffer now implements a true circular buffer with optimal O(1) performance for all operations!

---

## Summary of Manual Test Programs

This project includes four manual test programs for interactively testing the AnyBuffer adapter
implementations. Each program provides control bits for manual testing and status monitoring.

### SampleFifo - Bounded Queue Testing
**File**: POUs/SampleFifo.TcPOU
**Adapter**: FifoBuffer (bounded FIFO queue without overwrite)
**Buffer Size**: 3 elements (indices 0..2)
**Performance**: Push O(1), Pop O(n)

**Configuration**:
```iecst
fifo : FifoBuffer(anyBuffer, overwrite := FALSE, reversed := FALSE);
```

**Features**:
- Tests bounded queue behavior (rejects push when full)
- Optimized for frequent Push operations (O(1) constant time)
- Status info: isEmpty, isFull, elementCount, capacity
- Operation counters: pushCount, popCount, pushFailCount, popFailCount
- Auto-incrementing element IDs for easy tracking

**Manual Controls**:
- `bPush` - Push new element (fails when buffer is full)
- `bPop` - Pop oldest element (FIFO order)
- `bClear` - Clear all elements

**Testing Scenario**:
1. Push 3 elements → buffer becomes full
2. Try pushing 4th element → fails (pushFailCount increments)
3. Pop 1 element → creates space
4. Push again → now succeeds

### SampleLifo - Bounded Stack Testing
**File**: POUs/SampleLifo.TcPOU
**Adapter**: LifoBuffer (bounded LIFO/stack without overwrite)
**Buffer Size**: 3 elements (indices 0..2)
**Performance**: Push O(1), Pop O(1)

**Configuration**:
```iecst
lifo : LifoBuffer(anyBuffer, overwrite := FALSE, reversed := FALSE);
```

**Features**:
- Tests bounded stack behavior (rejects push when full)
- LIFO semantics: Last-In, First-Out (stack operations)
- Both Push and Pop are O(1) constant time operations
- Status info: isEmpty, isFull, elementCount, capacity
- Operation counters: pushCount, popCount, pushFailCount, popFailCount
- Auto-incrementing element IDs for easy tracking

**Manual Controls**:
- `bPush` - Push new element to top of stack (fails when buffer is full)
- `bPop` - Pop most recent element (LIFO order)
- `bClear` - Clear all elements

**Testing Scenario**:
1. Push elements with IDs 1, 2, 3 → buffer becomes full
2. Try pushing 4th element → fails (pushFailCount increments)
3. Pop element → returns ID 3 (last pushed, LIFO)
4. Pop again → returns ID 2 (second-to-last pushed)
5. Pop again → returns ID 1 (first pushed)
6. Observe: LIFO behavior - reverse order from FIFO

### SampleRing - Circular Buffer Testing
**File**: POUs/SampleRing.TcPOU
**Adapter**: RingBuffer (circular buffer with automatic overwrite)
**Buffer Size**: 5 elements (indices 0..4)
**Performance**: Push O(1), Pop O(1) - **No shifting operations!**

**Configuration**:
```iecst
ring : RingBuffer(anyBuffer, overwriteEnabled := TRUE);
```

**Features**:
- Tests circular buffer behavior (automatic overwrite of oldest)
- True O(1) performance using head/tail circular indexing
- No element shifting - direct memory access with WriteAtIndex
- Status info: isEmpty, isFull, elementCount, capacity, overwriteEnabled
- Operation counters: pushCount, popCount, pushFailCount, popFailCount, **overwriteCount**
- Buffer snapshot array for visualizing circular behavior
- Tracks how many times push triggered an overwrite

**Manual Controls**:
- `bPush` - Push new element (overwrites oldest when full)
- `bPop` - Pop oldest element
- `bClear` - Clear all elements
- `bToggleOverwrite` - Display toggle (informational only)

**Testing Scenario**:
1. Push 5 elements → buffer becomes full: [0, 1, 2, 3, 4]
2. Push 6th element (ID=5) → succeeds, removes 0: [1, 2, 3, 4, 5]
3. Push 7th element (ID=6) → succeeds, removes 1: [2, 3, 4, 5, 6]
4. Watch bufferSnapshot to observe elements cycling through
5. Pop retrieves current oldest (not original first element)

### SampleList - Directional Fill with Shift-Overwrite
**File**: POUs/SampleList.TcPOU
**Adapter**: List (configurable-direction FIFO with shift-overwrite)
**Buffer Size**: 5 elements (indices 0..4)

**Configuration**:
```iecst
list : List(anyBuffer, fillFromLeft := FALSE);  // Append mode (default)
```

**Features**:
- Tests directional fill behavior (append or prepend)
- Status info: isEmpty, isFull, elementCount, capacity, fillFromLeft
- Operation counters: pushCount, popCount, pushFailCount, popFailCount, **shiftOverwriteCount**
- Buffer snapshot array for visualizing shift behavior
- Direction info: fillDirectionInfo, pushPerformance strings
- Tracks shift-and-overwrite operations

**Manual Controls**:
- `bPush` - Push new element (shift-overwrites oldest when full)
- `bPop` - Pop oldest element (FIFO order)
- `bClear` - Clear all elements
- `bToggleFillDirection` - Display toggle (requires rebuild to change actual direction)

**Fill Direction Modes**:

**Mode A: fillFromLeft = FALSE (Append Mode - DEFAULT)**
- Push: Adds to end using AppendRight - O(1)
- Pop: Removes from front using PopLeft - O(n)
- Visual: `[oldest at 0] → [newer] → [newest at end]`
- Best for: Frequent pushes, infrequent pops

**Mode B: fillFromLeft = TRUE (Prepend Mode)**
- Push: Adds to front using AppendLeft - O(n)
- Pop: Removes from end using PopRight - O(1)
- Visual: `[newest at 0] ← [older] ← [oldest at end]`
- Best for: Frequent pops, infrequent pushes

**Testing Scenario (Append Mode)**:
1. Push 5 elements → buffer: [0, 1, 2, 3, 4] (IDs in order)
2. Push 6th element (ID=5) → shift-overwrite: [1, 2, 3, 4, 5] (0 removed from front)
3. Push 7th element (ID=6) → shift-overwrite: [2, 3, 4, 5, 6] (1 removed from front)
4. Pop → returns 2 (oldest remaining)
5. Observe: Push is fast O(1), Pop requires shifting O(n)

## Comparison Table

| Feature | SampleFifo | SampleLifo | SampleRing | SampleList |
|---------|------------|------------|------------|------------|
| **Adapter Type** | FifoBuffer | LifoBuffer | RingBuffer | List |
| **Buffer Size** | 3 elements | 3 elements | 5 elements | 5 elements |
| **Push Performance** | O(1) | O(1) | O(1) | O(1) or O(n) |
| **Pop Performance** | O(n) | O(1) | O(1) | O(1) or O(n) |
| **Semantic Order** | FIFO (queue) | LIFO (stack) | FIFO (circular) | FIFO (shift) |
| **Overwrite** | No (fails) | No (fails) | Yes (circular) | Yes (shift) |
| **Special Counter** | - | - | overwriteCount | shiftOverwriteCount |
| **Buffer Snapshot** | No | No | Yes | Yes |
| **Direction Config** | Fixed | Fixed | Fixed | Configurable |
| **Best for Testing** | Queue limits | Stack behavior | Circular behavior | Directional fill |

## Common Features

All four sample programs share:
- **ST_Element structure**: Simple struct with id (INT) and name (STRING)
- **Status display**: isEmpty, isFull, elementCount, capacity
- **Operation counters**: Track successful and failed push/pop operations
- **Persistent buffer**: Buffer array is PERSISTENT for observing data across PLC cycles
- **Auto-incrementing IDs**: Easy to track element insertion order

## Usage Instructions

1. **Add to task**: Ensure the desired sample program is called in MAIN or mapped to a task
2. **Online mode**: Go online with the PLC
3. **Watch variables**: Add program variables to watch list
4. **Set control bits**: Set bPush, bPop, or bClear to TRUE to trigger actions
5. **Observe behavior**: Watch counters, status, and bufferSnapshot (Ring/List) to understand behavior
6. **Test edge cases**: Try pushing to full buffer, popping from empty, etc.

## Test Data Structure

```iecst
TYPE ST_Element :
STRUCT
    id      : INT;      // Auto-incremented on each push
    name    : STRING;   // Format: 'element :X' where X is the id
END_STRUCT
END_TYPE
```
*)

SampleFifo();
SampleLifo();
SampleList();
SampleRing();

END_PROGRAM

// ---- _Mockups/AnyBuffer/SampleFifo.TcPOU
// Manual test program for FifoBuffer adapter functionality
PROGRAM SampleFifo
VAR
	fifo					: FifoBuffer(anyBuffer, FALSE, FALSE);	// no overwrite, not reversed

	firstRun				: BOOL := TRUE; // lazy firstrun
	elementPush				: ST_TEST_AnyBuffer_Element;
	elementPop				: ST_TEST_AnyBuffer_Element;

	// Manual control bits
	bPush					: BOOL;
	bPop					: BOOL;
	bClear					: BOOL;

	// Status information
	isEmpty					: BOOL;
	isFull					: BOOL;
	elementCount			: DINT;
	capacity				: DINT;

	// Operation counters
	pushCount				: UDINT;
	popCount				: UDINT;
	pushFailCount			: UDINT;
	popFailCount			: UDINT;
END_VAR

// Manual control actions
IF bClear			THEN
	bClear 			:= FALSE;
	fifo.Clear();
ELSIF bPush			THEN
	bPush 			:= FALSE;
	elementPush.id 		:= elementPush.id + 1;
	elementPush.name	:= concat('element :', TO_STRING(elementPush.id));
	IF fifo.Push(elementPush) THEN
		pushCount := pushCount + 1;
	ELSE
		pushFailCount := pushFailCount + 1;
	END_IF
ELSIF bPop			THEN
	bPop 			:= FALSE;
	IF fifo.Pop(elementPop) THEN
		popCount := popCount + 1;
	ELSE
		popFailCount := popFailCount + 1;
	END_IF
END_IF

// Update status information
isEmpty := fifo.isEmpty;
isFull := fifo.isFull;
elementCount := anyBuffer.Metadata.elementCount;
capacity := anyBuffer.Metadata.capacity;

END_PROGRAM

// ---- _Mockups/AnyBuffer/SampleLifo.TcPOU
// Manual test program for LifoBuffer adapter functionality
PROGRAM SampleLifo
VAR
	lifo					: LifoBuffer(anyBuffer, FALSE, FALSE);	// no overwrite, not reversed

	firstRun				: BOOL := TRUE; // lazy firstrun
	elementPush				: ST_TEST_AnyBuffer_Element;
	elementPop				: ST_TEST_AnyBuffer_Element;

	// Manual control bits
	bPush					: BOOL;
	bPop					: BOOL;
	bClear					: BOOL;

	// Status information
	isEmpty					: BOOL;
	isFull					: BOOL;
	elementCount			: DINT;
	capacity				: DINT;

	// Operation counters
	pushCount				: UDINT;
	popCount				: UDINT;
	pushFailCount			: UDINT;
	popFailCount			: UDINT;
END_VAR

// Manual control actions
IF bClear			THEN
	bClear 			:= FALSE;
	lifo.Clear();
ELSIF bPush			THEN
	bPush 			:= FALSE;
	elementPush.id 		:= elementPush.id + 1;
	elementPush.name	:= concat('element :', TO_STRING(elementPush.id));
	IF lifo.Push(elementPush) THEN
		pushCount := pushCount + 1;
	ELSE
		pushFailCount := pushFailCount + 1;
	END_IF
ELSIF bPop			THEN
	bPop 			:= FALSE;
	IF lifo.Pop(elementPop) THEN
		popCount := popCount + 1;
	ELSE
		popFailCount := popFailCount + 1;
	END_IF
END_IF

// Update status information
isEmpty := lifo.isEmpty;
isFull := lifo.isFull;
elementCount := anyBuffer.Metadata.elementCount;
capacity := anyBuffer.Metadata.capacity;

END_PROGRAM

// ---- _Mockups/AnyBuffer/SampleList.TcPOU
// Manual test program for List adapter functionality with directional fill and shift-overwrite
PROGRAM SampleList
VAR
	list					: ListBuffer(anyBuffer, FALSE);				// fillFromLeft=FALSE (append mode, default)

	firstRun				: BOOL := TRUE; // lazy firstrun
	elementPush				: ST_TEST_AnyBuffer_Element;
	elementPop				: ST_TEST_AnyBuffer_Element;

	// Manual control bits
	bPush					: BOOL;
	bPop					: BOOL;
	bClear					: BOOL;
	bToggleFillDirection	: BOOL;  // Toggle fill direction (note: requires reinit)

	// Status information
	isEmpty					: BOOL;
	isFull					: BOOL;
	elementCount			: DINT;
	capacity				: DINT;
	fillFromLeft			: BOOL := FALSE;  // Display current fill direction

	// Operation counters
	pushCount				: UDINT;
	popCount				: UDINT;
	pushFailCount			: UDINT;
	popFailCount			: UDINT;
	shiftOverwriteCount		: UDINT;  // Track how many times we pushed to full buffer (shift-overwrite)

	// Visual buffer state (for debugging)
	bufferSnapshot			: ARRAY[S_LL..S_UL] OF ST_TEST_AnyBuffer_Element;  // Copy of current buffer state

	// Fill direction info display
	fillDirectionInfo		: STRING := 'Fill from RIGHT (append)';  // Human-readable fill direction
	pushPerformance			: STRING := 'Push: O(1), Pop: O(n)';    // Performance characteristics
END_VAR
VAR CONSTANT
	LL						: INT := 0;
	UL						: INT := 4;  // Moderate buffer size to observe shift behavior
END_VAR

// Manual control actions
IF bClear			THEN
	bClear 			:= FALSE;
	list.Clear();
	shiftOverwriteCount := 0;  // Reset overwrite counter on clear
ELSIF bToggleFillDirection THEN
	bToggleFillDirection := FALSE;
	// Note: Fill direction is set at initialization and cannot be changed at runtime
	// This is just for demonstration - would need to recreate the List instance
	// For testing: manually change the list instantiation parameter and rebuild
	fillFromLeft := NOT fillFromLeft;
	IF fillFromLeft THEN
		fillDirectionInfo := 'Fill from LEFT (prepend)';
		pushPerformance := 'Push: O(n), Pop: O(1)';
	ELSE
		fillDirectionInfo := 'Fill from RIGHT (append)';
		pushPerformance := 'Push: O(1), Pop: O(n)';
	END_IF
ELSIF bPush			THEN
	bPush 			:= FALSE;
	elementPush.id 		:= elementPush.id + 1;
	elementPush.name	:= concat('element :', TO_STRING(elementPush.id));

	// Track if pushing to a full buffer (will trigger shift-and-overwrite)
	IF isFull THEN
		shiftOverwriteCount := shiftOverwriteCount + 1;
	END_IF

	IF list.Push(elementPush) THEN
		pushCount := pushCount + 1;
	ELSE
		pushFailCount := pushFailCount + 1;
	END_IF
ELSIF bPop			THEN
	bPop 			:= FALSE;
	IF list.Pop(elementPop) THEN
		popCount := popCount + 1;
	ELSE
		popFailCount := popFailCount + 1;
	END_IF
END_IF

// Update status information
isEmpty := list.isEmpty;
isFull := list.isFull;
elementCount := anyBuffer.Metadata.elementCount;
capacity := anyBuffer.Metadata.capacity;

// Update buffer snapshot for visualization
bufferSnapshot := buffer;

// Visual representation of buffer state
// When fillFromLeft=FALSE: [oldest at 0] -> [newer] -> [newest at end]
// When fillFromLeft=TRUE:  [newest at 0] <- [older] <- [oldest at end]

END_PROGRAM

// ---- _Mockups/AnyBuffer/SampleRing.TcPOU
// Manual test program for RingBuffer adapter functionality with circular overwrite
PROGRAM SampleRing
VAR
	ring					: RingBuffer(anyBuffer, TRUE);			// overwrite enabled (circular buffer mode)

	firstRun				: BOOL := TRUE; // lazy firstrun
	elementPush				: ST_TEST_AnyBuffer_Element;
	elementPop				: ST_TEST_AnyBuffer_Element;

	// Manual control bits
	bPush					: BOOL;
	bPop					: BOOL;
	bClear					: BOOL;
	bToggleOverwrite		: BOOL;  // Toggle overwrite mode on/off

	// Status information
	isEmpty					: BOOL;
	isFull					: BOOL;
	elementCount			: DINT;
	capacity				: DINT;
	overwriteEnabled		: BOOL := TRUE;  // Display current overwrite mode

	// Operation counters
	pushCount				: UDINT;
	popCount				: UDINT;
	pushFailCount			: UDINT;
	popFailCount			: UDINT;
	overwriteCount			: UDINT;  // Track how many times we pushed to a full buffer

	// Visual buffer state (for debugging)
	bufferSnapshot			: ARRAY[S_LL..S_UL] OF ST_TEST_AnyBuffer_Element;  // Copy of current buffer state
END_VAR
VAR CONSTANT
	LL						: INT := 0;
	UL						: INT := 4;  // Slightly larger buffer to see circular behavior
END_VAR

// Manual control actions
IF bClear			THEN
	bClear 			:= FALSE;
	ring.Clear();
	overwriteCount := 0;  // Reset overwrite counter on clear
ELSIF bToggleOverwrite THEN
	bToggleOverwrite := FALSE;
	// Note: Overwrite mode is set at initialization and cannot be changed at runtime
	// This is just for demonstration - would need to recreate the RingBuffer instance
	// overwriteEnabled := NOT overwriteEnabled;
ELSIF bPush			THEN
	bPush 			:= FALSE;
	elementPush.id 		:= elementPush.id + 1;
	elementPush.name	:= concat('element :', TO_STRING(elementPush.id));

	// Track if pushing to a full buffer (will trigger overwrite in circular mode)
	IF isFull AND overwriteEnabled THEN
		overwriteCount := overwriteCount + 1;
	END_IF

	IF ring.Push(elementPush) THEN
		pushCount := pushCount + 1;
	ELSE
		pushFailCount := pushFailCount + 1;
	END_IF
ELSIF bPop			THEN
	bPop 			:= FALSE;
	IF ring.Pop(elementPop) THEN
		popCount := popCount + 1;
	ELSE
		popFailCount := popFailCount + 1;
	END_IF
END_IF

// Update status information
isEmpty := ring.isEmpty;
isFull := ring.isFull;
elementCount := anyBuffer.Metadata.elementCount;
capacity := anyBuffer.Metadata.capacity;

// Update buffer snapshot for visualization
bufferSnapshot := buffer;

END_PROGRAM

// ---- UnitTests/AnyBuffer/TEST_AnyBuffer_Clear.TcPOU
PROGRAM TEST_AnyBuffer_Clear

ClearsAllElements();
ResetsElementCount();
ResetsAllMetadata();
ReturnsTrue();
ClearEmptyBuffer();
ClearAfterPush();
ClearAfterPop();
MultipleClearCalls();
ClearFullBuffer();
ClearPartialBuffer();
PreservesConfiguration();
CanReuseAfterClear();

// Buffer can be reused (push/pop) immediately after Clear
METHOD CanReuseAfterClear
VAR
	ReturnedElement : DINT;
END_VAR
IF TestSuite.Test(__POUNAME()).ExecuteTest() THEN
	// Arrange - Fill and clear buffer
	fbAnyBuffer.Clear();
	testElement := DINT#100;
	fbAnyBuffer.PushLeft(element := testElement);
	fbAnyBuffer.Clear();

	// Act - Reuse buffer immediately after clear
	testElement := DINT#200;
	Success := fbAnyBuffer.PushLeft(element := testElement);
	TestSuite.Test(__POUNAME()).AssertEqual(TEST_BOOL_TRUE, Success);

	testElement := DINT#300;
	Success := fbAnyBuffer.PushLeft(element := testElement);
	TestSuite.Test(__POUNAME()).AssertEqual(TEST_BOOL_TRUE, Success);

	Success := fbAnyBuffer.PopLeft(element := ReturnedElement);
	TestSuite.Test(__POUNAME()).AssertEqual(TEST_BOOL_TRUE, Success);

	// Assert - Buffer works correctly after clear
	TEST_DINT := 300;
	TestSuite.Test(__POUNAME()).AssertEqual(TEST_DINT, ReturnedElement);
	TEST_DINT := 1;
	TestSuite.Test(__POUNAME()).AssertEqual(TEST_DINT, fbAnyBuffer.Metadata.elementCount);
END_IF
END_METHOD

